C01835=1141.275,213.757,-64.467,-177.986,7.593,148.858
C01836=1141.271,214.006,-64.493,-177.983,7.596,148.857
C01837=1141.266,214.256,-64.518,-177.981,7.599,148.857
C01838=1141.261,214.504,-64.544,-177.977,7.602,148.857
C01839=1141.257,214.753,-64.569,-177.975,7.604,148.857
C01840=1141.253,215.001,-64.593,-177.972,7.607,148.857
C01841=1141.248,215.250,-64.619,-177.969,7.610,148.857
C01842=1141.243,215.498,-64.644,-177.966,7.612,148.856
C01843=1141.239,215.747,-64.670,-177.963,7.615,148.856
C01844=1141.234,215.995,-64.695,-177.961,7.617,148.856
C01845=1141.230,216.245,-64.720,-177.958,7.620,148.856
C01846=1141.225,216.494,-64.746,-177.955,7.623,148.856
C01847=1141.221,216.741,-64.770,-177.952,7.626,148.856
C01848=1141.217,216.991,-64.796,-177.950,7.628,148.856
C01849=1141.212,217.239,-64.821,-177.947,7.631,148.855
C01850=1141.208,217.488,-64.847,-177.944,7.633,148.855
C01851=1141.203,217.737,-64.872,-177.941,7.636,148.855
C01852=1141.198,217.985,-64.897,-177.938,7.639,148.855
C01853=1141.194,218.234,-64.923,-177.936,7.641,148.855
C01854=1141.189,218.482,-64.948,-177.933,7.644,148.854
C01855=1141.185,218.731,-64.974,-177.930,7.646,148.854
C01856=1141.181,218.980,-64.999,-177.927,7.649,148.854
C01857=1141.176,219.228,-65.024,-177.924,7.652,148.854
C01858=1141.172,219.477,-65.050,-177.922,7.654,148.854
C01859=1141.167,219.726,-65.076,-177.919,7.657,148.854
C01860=1141.162,219.974,-65.101,-177.916,7.660,148.854
C01861=1141.158,220.223,-65.127,-177.913,7.663,148.854
C01862=1141.154,220.472,-65.153,-177.911,7.666,148.853
C01863=1141.149,220.720,-65.177,-177.907,7.668,148.853
C01864=1141.145,220.969,-65.203,-177.905,7.670,148.853
C01865=1141.140,221.218,-65.229,-177.902,7.673,148.853
C01866=1141.136,221.466,-65.254,-177.899,7.676,148.853
C01867=1141.131,221.715,-65.280,-177.897,7.679,148.853
C01868=1141.127,221.964,-65.306,-177.894,7.682,148.853
C01869=1141.123,222.213,-65.332,-177.891,7.685,148.852
C01870=1141.118,222.461,-65.357,-177.888,7.687,148.852
C01871=1141.114,222.709,-65.383,-177.886,7.690,148.852
C01872=1141.109,222.959,-65.409,-177.883,7.692,148.852
C01873=1141.104,223.207,-65.434,-177.880,7.695,148.852
C01874=1141.100,223.456,-65.460,-177.877,7.698,148.852
C01875=1141.096,223.704,-65.486,-177.874,7.701,148.852
C01876=1141.091,223.953,-65.512,-177.872,7.703,148.851
C01877=1141.087,224.201,-65.537,-177.869,7.706,148.851
C01878=1141.083,224.449,-65.564,-177.866,7.709,148.851
C01879=1141.078,224.699,-65.590,-177.863,7.712,148.851
C01880=1141.074,224.947,-65.616,-177.860,7.714,148.851
C01881=1141.069,225.195,-65.641,-177.857,7.717,148.851
C01882=1141.064,225.444,-65.667,-177.854,7.720,148.851
C01883=1141.060,225.693,-65.693,-177.852,7.722,148.851
C01884=1141.055,225.942,-65.719,-177.849,7.725,148.850
C01885=1141.051,226.190,-65.745,-177.847,7.728,148.850
C01886=1141.047,226.438,-65.771,-177.843,7.731,148.850
C01887=1141.042,226.687,-65.796,-177.841,7.733,148.850
C01888=1141.037,226.936,-65.823,-177.838,7.736,148.850
C01889=1141.033,227.185,-65.849,-177.835,7.739,148.850
C01890=1141.029,227.433,-65.875,-177.833,7.741,148.850
C01891=1141.024,227.681,-65.900,-177.830,7.744,148.850
C01892=1141.019,227.931,-65.927,-177.827,7.747,148.850
C01893=1141.015,228.179,-65.953,-177.824,7.750,148.849
C01894=1141.011,228.428,-65.979,-177.821,7.753,148.849
C01895=1141.006,228.677,-66.005,-177.818,7.756,148.849
C01896=1141.002,228.925,-66.032,-177.815,7.759,148.849
C01897=1140.998,229.174,-66.058,-177.813,7.761,148.849
C01898=1140.993,229.422,-66.084,-177.810,7.764,148.849
C01899=1140.989,229.670,-66.110,-177.808,7.766,148.849
C01900=1140.984,229.919,-66.136,-177.805,7.769,148.849
C01901=1140.979,230.168,-66.162,-177.802,7.772,148.848
C01902=1140.976,230.416,-66.189,-177.799,7.775,148.848
C01903=1140.971,230.665,-66.214,-177.796,7.778,148.848
C01904=1140.967,230.914,-66.241,-177.793,7.781,148.848
C01905=1140.962,231.162,-66.267,-177.790,7.784,148.848
C01906=1140.958,231.411,-66.294,-177.788,7.786,148.848
C01907=1140.953,231.659,-66.320,-177.785,7.789,148.848
C01908=1140.949,231.907,-66.346,-177.783,7.791,148.848
C01909=1140.944,232.156,-66.372,-177.780,7.794,148.848
C01910=1140.940,232.405,-66.399,-177.777,7.797,148.847
C01911=1140.935,232.654,-66.425,-177.774,7.800,148.847
C01912=1140.931,232.902,-66.452,-177.771,7.803,148.847
C01913=1140.926,233.151,-66.478,-177.768,7.806,148.847
C01914=1140.922,233.399,-66.504,-177.765,7.809,148.847
C01915=1140.918,233.648,-66.532,-177.763,7.812,148.847
C01916=1140.914,233.896,-66.557,-177.760,7.814,148.847
C01917=1140.909,234.145,-66.584,-177.757,7.817,148.847
C01918=1140.905,234.394,-66.610,-177.754,7.820,148.847
C01919=1140.900,234.642,-66.637,-177.752,7.822,148.846
C01920=1140.896,234.890,-66.664,-177.749,7.825,148.846
C01921=1140.891,235.163,-66.692,-177.746,7.829,148.846
C01922=1140.886,235.434,-66.722,-177.743,7.832,148.846
C01923=1140.882,235.706,-66.751,-177.740,7.834,148.846
C01924=1140.877,235.978,-66.780,-177.736,7.838,148.846
C01925=1140.872,236.227,-66.806,-177.733,7.841,148.846
C01926=1140.868,236.475,-66.833,-177.731,7.843,148.846
C01927=1140.863,236.724,-66.860,-177.728,7.846,148.846
C01928=1140.859,236.972,-66.886,-177.726,7.849,148.846
C01929=1140.854,237.221,-66.913,-177.723,7.852,148.845
C01930=1140.850,237.469,-66.940,-177.720,7.855,148.845
C01931=1140.846,237.718,-66.966,-177.717,7.858,148.845
C01932=1140.841,237.966,-66.993,-177.714,7.861,148.845
C01933=1140.836,238.215,-67.020,-177.712,7.864,148.845
C01934=1140.832,238.463,-67.046,-177.709,7.867,148.845
C01935=1140.827,238.712,-67.073,-177.706,7.869,148.845
C01936=1140.823,238.961,-67.101,-177.703,7.872,148.845
C01937=1140.819,239.209,-67.127,-177.701,7.875,148.845
C01938=1140.815,239.458,-67.154,-177.698,7.878,148.845
C01939=1140.810,239.706,-67.181,-177.695,7.881,148.845
C01940=1140.806,239.954,-67.208,-177.692,7.884,148.845
C01941=1140.802,240.203,-67.235,-177.689,7.887,148.844
C01942=1140.797,240.451,-67.262,-177.687,7.890,148.844
C01943=1140.792,240.700,-67.289,-177.684,7.893,148.844
C01944=1140.788,240.948,-67.315,-177.681,7.896,148.844
C01945=1140.784,241.197,-67.342,-177.678,7.899,148.844
C01946=1140.780,241.446,-67.370,-177.675,7.902,148.844
C01947=1140.775,241.694,-67.397,-177.673,7.904,148.844
C01948=1140.771,241.943,-67.423,-177.670,7.907,148.844
C01949=1140.766,242.191,-67.450,-177.668,7.909,148.844
C01950=1140.762,242.440,-67.477,-177.665,7.912,148.844
C01951=1140.757,242.688,-67.505,-177.662,7.915,148.844
C01952=1140.752,242.937,-67.532,-177.659,7.918,148.844
C01953=1140.749,243.185,-67.558,-177.656,7.921,148.843
C01954=1140.744,243.434,-67.586,-177.654,7.924,148.843
C01955=1140.740,243.682,-67.613,-177.651,7.927,148.843
C01956=1140.735,243.930,-67.640,-177.648,7.930,148.843
C01957=1140.731,244.179,-67.667,-177.645,7.933,148.843
C01958=1140.727,244.428,-67.695,-177.642,7.936,148.843
C01959=1140.722,244.676,-67.722,-177.640,7.939,148.843
C01960=1140.718,244.925,-67.748,-177.637,7.942,148.843
C01961=1140.714,245.172,-67.776,-177.634,7.944,148.843
C01962=1140.709,245.421,-67.803,-177.631,7.947,148.843
C01963=1140.705,245.670,-67.831,-177.628,7.950,148.843
C01964=1140.700,245.919,-67.858,-177.626,7.953,148.843
C01965=1140.696,246.167,-67.885,-177.623,7.956,148.843
C01966=1140.691,246.415,-67.913,-177.620,7.959,148.843
C01967=1140.687,246.664,-67.940,-177.617,7.962,148.842
C01968=1140.683,246.913,-67.967,-177.614,7.965,148.842
C01969=1140.678,247.161,-67.995,-177.612,7.968,148.842
C01970=1140.674,247.409,-68.022,-177.609,7.971,148.842
C01971=1140.670,247.658,-68.050,-177.606,7.974,148.842
C01972=1140.665,247.906,-68.077,-177.603,7.977,148.842
C01973=1140.661,248.155,-68.104,-177.600,7.979,148.842
C01974=1140.656,248.403,-68.132,-177.598,7.982,148.842
C01975=1140.652,248.652,-68.159,-177.595,7.985,148.842
C01976=1140.648,248.900,-68.186,-177.592,7.989,148.842
C01977=1140.643,249.148,-68.214,-177.590,7.991,148.842
C01978=1140.639,249.397,-68.242,-177.587,7.994,148.842
C01979=1140.635,249.645,-68.269,-177.584,7.997,148.842
C01980=1140.630,249.894,-68.296,-177.581,8.000,148.842
C01981=1140.626,250.142,-68.324,-177.578,8.004,148.842
C01982=1140.622,250.391,-68.352,-177.575,8.007,148.842
C01983=1140.617,250.639,-68.379,-177.572,8.010,148.842
C01984=1140.613,250.887,-68.406,-177.570,8.013,148.841
C01985=1140.608,251.136,-68.435,-177.567,8.016,148.841
C01986=1140.604,251.385,-68.462,-177.564,8.019,148.841
C01987=1140.600,251.633,-68.490,-177.561,8.021,148.841
C01988=1140.596,251.881,-68.518,-177.559,8.025,148.841
C01989=1140.591,252.129,-68.545,-177.556,8.028,148.841
C01990=1140.587,252.378,-68.573,-177.553,8.031,148.841
C01991=1140.583,252.626,-68.601,-177.550,8.034,148.841
C01992=1140.577,252.875,-68.629,-177.548,8.036,148.841
C01993=1140.574,253.123,-68.657,-177.545,8.039,148.841
C01994=1140.569,253.372,-68.684,-177.542,8.042,148.841
C01995=1140.565,253.620,-68.712,-177.539,8.045,148.841
C01996=1140.561,253.868,-68.740,-177.536,8.048,148.841
C01997=1140.556,254.116,-68.768,-177.534,8.051,148.841
C01998=1140.552,254.366,-68.796,-177.531,8.054,148.841
C01999=1140.547,254.614,-68.824,-177.529,8.057,148.841
C02000=1140.544,254.862,-68.852,-177.526,8.060,148.841
C02001=1140.539,255.110,-68.879,-177.523,8.063,148.841
C02002=1140.534,255.359,-68.907,-177.520,8.066,148.841
C02003=1140.530,255.607,-68.935,-177.517,8.070,148.841
C02004=1140.526,255.855,-68.963,-177.514,8.073,148.841
C02005=1140.521,256.104,-68.992,-177.512,8.076,148.841
C02006=1140.517,256.352,-69.020,-177.509,8.079,148.841
C02007=1140.513,256.601,-69.047,-177.506,8.082,148.841
C02008=1140.508,256.849,-69.075,-177.503,8.085,148.840
C02009=1140.504,257.098,-69.103,-177.500,8.088,148.840
C02010=1140.500,257.346,-69.131,-177.498,8.090,148.840
C02011=1140.495,257.595,-69.160,-177.495,8.093,148.840
C02012=1140.491,257.843,-69.188,-177.493,8.097,148.840
C02013=1140.487,258.091,-69.216,-177.490,8.100,148.840
C02014=1140.482,258.339,-69.244,-177.487,8.102,148.840
C02015=1140.478,258.588,-69.272,-177.484,8.105,148.840
C02016=1140.474,258.836,-69.300,-177.481,8.109,148.840
C02017=1140.469,259.085,-69.329,-177.478,8.112,148.840
C02018=1140.465,259.333,-69.357,-177.476,8.115,148.840
C02019=1140.461,259.581,-69.385,-177.473,8.118,148.840
C02020=1140.456,259.829,-69.413,-177.470,8.121,148.840
C02021=1140.452,260.078,-69.441,-177.467,8.124,148.840
C02022=1140.447,260.326,-69.470,-177.464,8.127,148.840
C02023=1140.444,260.575,-69.498,-177.462,8.130,148.840
C02024=1140.439,260.823,-69.526,-177.459,8.133,148.840
C02025=1140.434,261.097,-69.557,-177.456,8.137,148.840
C02026=1140.429,261.371,-69.589,-177.453,8.140,148.840
C02027=1140.425,261.643,-69.620,-177.450,8.144,148.840
C02028=1140.420,261.918,-69.652,-177.447,8.146,148.840
C02029=1140.416,262.165,-69.679,-177.444,8.149,148.840
C02030=1140.411,262.414,-69.708,-177.441,8.153,148.840
C02031=1140.407,262.662,-69.736,-177.439,8.156,148.840
C02032=1140.403,262.911,-69.765,-177.436,8.159,148.840
C02033=1140.399,263.159,-69.794,-177.433,8.162,148.840
C02034=1140.394,263.407,-69.822,-177.430,8.165,148.840
C02035=1140.390,263.656,-69.850,-177.428,8.168,148.840
C02036=1140.385,263.903,-69.879,-177.425,8.171,148.840
C02037=1140.381,264.152,-69.907,-177.422,8.174,148.840
C02038=1140.377,264.401,-69.936,-177.419,8.178,148.840
C02039=1140.372,264.649,-69.964,-177.417,8.181,148.840
C02040=1140.368,264.897,-69.993,-177.414,8.184,148.840
C02041=1140.364,265.146,-70.022,-177.411,8.187,148.840
C02042=1140.359,265.394,-70.050,-177.408,8.190,148.840
C02043=1140.355,265.642,-70.079,-177.406,8.193,148.840
C02044=1140.351,265.891,-70.108,-177.403,8.196,148.840
C02045=1140.347,266.138,-70.136,-177.400,8.199,148.840
C02046=1140.342,266.387,-70.165,-177.397,8.203,148.840
C02047=1140.338,266.636,-70.194,-177.395,8.206,148.840
C02048=1140.334,266.883,-70.222,-177.392,8.209,148.840
C02049=1140.329,267.132,-70.251,-177.389,8.212,148.840
C02050=1140.325,267.380,-70.281,-177.386,8.215,148.840
C02051=1140.320,267.629,-70.309,-177.384,8.218,148.840
C02052=1140.317,267.877,-70.338,-177.381,8.221,148.840
C02053=1140.312,268.125,-70.367,-177.378,8.225,148.840
C02054=1140.308,268.374,-70.396,-177.375,8.228,148.840
C02055=1140.303,268.622,-70.424,-177.372,8.231,148.840
C02056=1140.299,268.870,-70.453,-177.370,8.234,148.840
C02057=1140.295,269.119,-70.482,-177.367,8.237,148.840
C02058=1140.291,269.367,-70.511,-177.365,8.240,148.840
C02059=1140.286,269.615,-70.540,-177.362,8.243,148.840
C02060=1140.282,269.863,-70.569,-177.358,8.247,148.840
C02061=1140.278,270.112,-70.597,-177.356,8.250,148.840
C02062=1140.274,270.360,-70.627,-177.353,8.253,148.840
C02063=1140.269,270.608,-70.656,-177.350,8.256,148.840
C02064=1140.264,270.857,-70.685,-177.348,8.259,148.840
C02065=1140.261,271.105,-70.714,-177.345,8.262,148.840
C02066=1140.257,271.353,-70.743,-177.342,8.266,148.840
C02067=1140.252,271.602,-70.772,-177.339,8.269,148.840
C02068=1140.247,271.849,-70.801,-177.337,8.272,148.840
C02069=1140.243,272.098,-70.830,-177.334,8.275,148.840
C02070=1140.239,272.346,-70.860,-177.331,8.278,148.840
C02071=1140.235,272.595,-70.888,-177.329,8.281,148.840
C02072=1140.231,272.843,-70.917,-177.326,8.285,148.840
C02073=1140.226,273.090,-70.946,-177.323,8.288,148.840
C02074=1140.222,273.339,-70.976,-177.320,8.291,148.840
C02075=1140.218,273.588,-71.005,-177.318,8.294,148.840
C02076=1140.213,273.836,-71.034,-177.315,8.297,148.840
C02077=1140.209,274.084,-71.063,-177.312,8.301,148.840
C02078=1140.205,274.332,-71.093,-177.309,8.304,148.840
C02079=1140.201,274.581,-71.122,-177.306,8.307,148.840
C02080=1140.196,274.828,-71.151,-177.304,8.310,148.840
C02081=1140.192,275.076,-71.181,-177.301,8.313,148.840
C02082=1140.187,275.325,-71.210,-177.298,8.316,148.840
C02083=1140.183,275.574,-71.239,-177.296,8.320,148.840
C02084=1140.179,275.822,-71.269,-177.293,8.323,148.840
C02085=1140.175,276.070,-71.298,-177.290,8.326,148.840
C02086=1140.171,276.318,-71.327,-177.288,8.329,148.840
C02087=1140.167,276.567,-71.357,-177.285,8.332,148.840
C02088=1140.162,276.815,-71.386,-177.281,8.336,148.840
C02089=1140.158,277.063,-71.416,-177.279,8.339,148.841
C02090=1140.153,277.311,-71.445,-177.276,8.342,148.840
C02091=1140.149,277.559,-71.474,-177.274,8.345,148.841
C02092=1140.145,277.807,-71.504,-177.271,8.349,148.841
C02093=1140.141,278.056,-71.533,-177.268,8.352,148.841
C02094=1140.137,278.304,-71.563,-177.265,8.355,148.841
C02095=1140.133,278.552,-71.592,-177.263,8.358,148.841
C02096=1140.129,278.800,-71.622,-177.260,8.361,148.841
C02097=1140.124,279.048,-71.652,-177.257,8.365,148.841
C02098=1140.120,279.297,-71.682,-177.254,8.368,148.841
C02099=1140.115,279.545,-71.711,-177.252,8.371,148.841
C02100=1140.111,279.793,-71.741,-177.249,8.374,148.841
C02101=1140.107,280.041,-71.770,-177.247,8.377,148.841
C02102=1140.103,280.290,-71.800,-177.243,8.381,148.841
C02103=1140.099,280.537,-71.830,-177.241,8.384,148.841
C02104=1140.094,280.786,-71.860,-177.238,8.387,148.841
C02105=1140.090,281.034,-71.889,-177.235,8.390,148.841
C02106=1140.086,281.282,-71.919,-177.233,8.394,148.841
C02107=1140.082,281.530,-71.949,-177.230,8.397,148.841
C02108=1140.078,281.778,-71.978,-177.227,8.401,148.841
C02109=1140.073,282.027,-72.008,-177.225,8.403,148.841
C02110=1140.068,282.275,-72.038,-177.222,8.408,148.842
C02111=1140.065,282.523,-72.068,-177.219,8.410,148.841
C02112=1140.060,282.771,-72.098,-177.216,8.413,148.841
C02113=1140.056,283.020,-72.128,-177.214,8.417,148.842
C02114=1140.052,283.267,-72.158,-177.210,8.420,148.842
C02115=1140.047,283.516,-72.187,-177.208,8.424,148.842
C02116=1140.043,283.764,-72.217,-177.205,8.427,148.842
C02117=1140.039,284.012,-72.247,-177.203,8.430,148.842
C02118=1140.035,284.261,-72.277,-177.200,8.434,148.842
C02119=1140.031,284.508,-72.307,-177.197,8.437,148.842
C02120=1140.026,284.757,-72.337,-177.194,8.440,148.842
C02121=1140.022,285.005,-72.368,-177.192,8.443,148.842
C02122=1140.018,285.253,-72.397,-177.189,8.447,148.842
C02123=1140.014,285.501,-72.428,-177.186,8.450,148.842
C02124=1140.009,285.749,-72.457,-177.184,8.453,148.842
C02125=1140.005,285.997,-72.488,-177.181,8.456,148.842
C02126=1140.001,286.245,-72.518,-177.178,8.460,148.842
C02127=1139.997,286.493,-72.548,-177.176,8.463,148.843
C02128=1139.992,286.742,-72.578,-177.173,8.466,148.843
C02129=1139.988,287.017,-72.611,-177.170,8.470,148.843
C02130=1139.983,287.293,-72.644,-177.166,8.474,148.843
C02131=1139.978,287.568,-72.678,-177.164,8.477,148.843
C02132=1139.974,287.844,-72.712,-177.161,8.481,148.843
C02133=1139.969,288.092,-72.742,-177.158,8.484,148.843
C02134=1139.965,288.340,-72.772,-177.155,8.488,148.843
C02135=1139.961,288.589,-72.803,-177.153,8.491,148.843
C02136=1139.957,288.837,-72.833,-177.150,8.494,148.843
C02137=1139.952,289.085,-72.864,-177.147,8.498,148.843
C02138=1139.949,289.332,-72.894,-177.144,8.501,148.843
C02139=1139.944,289.581,-72.924,-177.142,8.504,148.844
C02140=1139.940,289.829,-72.954,-177.139,8.507,148.843
C02141=1139.936,290.077,-72.985,-177.136,8.511,148.844
C02142=1139.932,290.325,-73.015,-177.133,8.514,148.844
C02143=1139.927,290.574,-73.045,-177.131,8.518,148.844
C02144=1139.923,290.821,-73.075,-177.128,8.522,148.844
C02145=1139.919,291.070,-73.107,-177.125,8.525,148.844
C02146=1139.915,291.318,-73.137,-177.123,8.528,148.844
C02147=1139.911,291.565,-73.168,-177.120,8.532,148.844
C02148=1139.906,291.814,-73.197,-177.117,8.535,148.844
C02149=1139.902,292.062,-73.228,-177.114,8.538,148.844
C02150=1139.898,292.310,-73.259,-177.112,8.541,148.844
C02151=1139.894,292.558,-73.289,-177.109,8.545,148.845
C02152=1139.889,292.806,-73.320,-177.106,8.548,148.845
C02153=1139.886,293.054,-73.350,-177.104,8.551,148.845
C02154=1139.881,293.302,-73.381,-177.101,8.555,148.845
C02155=1139.877,293.550,-73.412,-177.098,8.558,148.845
C02156=1139.874,293.799,-73.442,-177.096,8.562,148.845
C02157=1139.869,294.047,-73.473,-177.093,8.565,148.845
C02158=1139.864,294.294,-73.504,-177.090,8.569,148.845
C02159=1139.861,294.543,-73.534,-177.088,8.571,148.845
C02160=1139.856,294.791,-73.565,-177.085,8.576,148.845
C02161=1139.852,295.039,-73.596,-177.082,8.579,148.846
C02162=1139.848,295.286,-73.626,-177.080,8.582,148.846
C02163=1139.844,295.535,-73.657,-177.077,8.586,148.846
C02164=1139.839,295.783,-73.688,-177.074,8.589,148.846
C02165=1139.835,296.032,-73.719,-177.071,8.592,148.846
C02166=1139.831,296.279,-73.749,-177.069,8.596,148.846
C02167=1139.827,296.527,-73.780,-177.066,8.599,148.846
C02168=1139.823,296.776,-73.811,-177.063,8.602,148.846
C02169=1139.818,297.023,-73.843,-177.060,8.606,148.846
C02170=1139.815,297.271,-73.873,-177.058,8.609,148.846
C02171=1139.811,297.520,-73.904,-177.055,8.612,148.847
C02172=1139.806,297.768,-73.935,-177.052,8.617,148.847
C02173=1139.801,298.016,-73.966,-177.050,8.620,148.847
C02174=1139.797,298.264,-73.997,-177.047,8.623,148.847
C02175=1139.794,298.511,-74.028,-177.044,8.627,148.847
C02176=1139.790,298.760,-74.059,-177.042,8.630,148.847
C02177=1139.785,299.008,-74.089,-177.039,8.633,148.847
C02178=1139.781,299.256,-74.120,-177.036,8.637,148.847
C02179=1139.777,299.504,-74.152,-177.034,8.640,148.848
C02180=1139.772,299.752,-74.183,-177.031,8.643,148.848
C02181=1139.768,300.000,-74.214,-177.028,8.647,148.848
C02182=1139.764,300.248,-74.245,-177.026,8.651,148.848
C02183=1139.761,300.496,-74.276,-177.023,8.654,148.848
C02184=1139.756,300.744,-74.307,-177.020,8.658,148.848
C02185=1139.752,300.992,-74.339,-177.018,8.661,148.848
C02186=1139.748,301.240,-74.369,-177.015,8.665,148.848
C02187=1139.743,301.487,-74.401,-177.012,8.668,148.849
C02188=1139.739,301.736,-74.432,-177.010,8.671,148.849
C02189=1139.735,301.984,-74.463,-177.007,8.675,148.849
C02190=1139.731,302.232,-74.495,-177.004,8.678,148.849
C02191=1139.726,302.480,-74.525,-177.001,8.682,148.849
C02192=1139.723,302.728,-74.557,-176.999,8.685,148.849
C02193=1139.718,302.976,-74.588,-176.997,8.689,148.849
C02194=1139.714,303.224,-74.620,-176.993,8.692,148.849
C02195=1139.710,303.472,-74.651,-176.991,8.696,148.850
C02196=1139.706,303.720,-74.682,-176.988,8.699,148.850
C02197=1139.701,303.968,-74.713,-176.986,8.703,148.850
C02198=1139.698,304.216,-74.745,-176.983,8.706,148.850
C02199=1139.693,304.464,-74.776,-176.980,8.710,148.850
C02200=1139.689,304.712,-74.808,-176.977,8.713,148.850
C02201=1139.685,304.959,-74.839,-176.975,8.717,148.851
C02202=1139.680,305.208,-74.871,-176.972,8.720,148.851
C02203=1139.676,305.456,-74.902,-176.969,8.724,148.851
C02204=1139.672,305.704,-74.934,-176.967,8.728,148.851
C02205=1139.668,305.952,-74.965,-176.964,8.731,148.851
C02206=1139.664,306.200,-74.997,-176.962,8.734,148.851
C02207=1139.660,306.448,-75.029,-176.958,8.738,148.851
C02208=1139.656,306.696,-75.059,-176.956,8.741,148.852
C02209=1139.652,306.944,-75.091,-176.953,8.745,148.852
C02210=1139.647,307.191,-75.123,-176.951,8.749,148.852
C02211=1139.643,307.440,-75.154,-176.949,8.752,148.852
C02212=1139.639,307.688,-75.186,-176.945,8.756,148.852
C02213=1139.635,307.935,-75.218,-176.943,8.759,148.852
C02214=1139.631,308.183,-75.250,-176.940,8.763,148.852
C02215=1139.628,308.432,-75.281,-176.938,8.766,148.853
C02216=1139.622,308.680,-75.313,-176.935,8.770,148.853
C02217=1139.618,308.928,-75.345,-176.932,8.773,148.853
C02218=1139.614,309.175,-75.376,-176.929,8.776,148.853
C02219=1139.610,309.423,-75.408,-176.927,8.780,148.853
C02220=1139.606,309.672,-75.440,-176.924,8.784,148.853
C02221=1139.602,309.919,-75.472,-176.921,8.788,148.854
C02222=1139.598,310.167,-75.504,-176.919,8.791,148.854
C02223=1139.594,310.415,-75.536,-176.916,8.795,148.854
C02224=1139.589,310.663,-75.568,-176.914,8.798,148.854
C02225=1139.586,310.911,-75.600,-176.911,8.802,148.854
C02226=1139.582,311.159,-75.631,-176.908,8.805,148.854
C02227=1139.577,311.407,-75.662,-176.906,8.809,148.855
C02228=1139.573,311.655,-75.695,-176.903,8.813,148.855
C02229=1139.569,311.903,-75.726,-176.900,8.816,148.855
C02230=1139.565,312.150,-75.759,-176.897,8.820,148.855
C02231=1139.561,312.398,-75.791,-176.895,8.823,148.855
C02232=1139.557,312.646,-75.823,-176.892,8.827,148.856
C02233=1139.552,312.925,-75.858,-176.890,8.831,148.856
C02234=1139.547,313.202,-75.894,-176.887,8.835,148.856
C02235=1139.543,313.481,-75.931,-176.884,8.838,148.856
C02236=1139.538,313.758,-75.966,-176.881,8.843,148.856
C02237=1139.534,314.007,-75.999,-176.878,8.847,148.857
C02238=1139.530,314.254,-76.030,-176.875,8.850,148.857
C02239=1139.526,314.501,-76.063,-176.872,8.854,148.857
C02240=1139.522,314.750,-76.095,-176.870,8.857,148.857
C02241=1139.518,314.998,-76.127,-176.867,8.861,148.857
C02242=1139.513,315.245,-76.159,-176.865,8.864,148.858
C02243=1139.509,315.493,-76.191,-176.862,8.869,148.858
C02244=1139.505,315.741,-76.224,-176.860,8.872,148.858
C02245=1139.502,315.989,-76.256,-176.857,8.876,148.858
C02246=1139.497,316.238,-76.288,-176.854,8.879,148.858
C02247=1139.493,316.485,-76.320,-176.851,8.883,148.859
C02248=1139.489,316.733,-76.353,-176.849,8.886,148.859
C02249=1139.485,316.981,-76.385,-176.846,8.891,148.859
C02250=1139.481,317.229,-76.417,-176.844,8.894,148.859
C02251=1139.477,317.476,-76.450,-176.841,8.898,148.859
C02252=1139.472,317.724,-76.482,-176.838,8.901,148.860
C02253=1139.469,317.971,-76.514,-176.836,8.904,148.860
C02254=1139.464,318.220,-76.547,-176.833,8.908,148.860
C02255=1139.461,318.468,-76.579,-176.831,8.912,148.860
C02256=1139.456,318.716,-76.612,-176.828,8.916,148.860
C02257=1139.453,318.964,-76.644,-176.826,8.919,148.861
C02258=1139.449,319.211,-76.677,-176.823,8.923,148.861
C02259=1139.444,319.459,-76.709,-176.820,8.926,148.861
C02260=1139.440,319.706,-76.741,-176.817,8.930,148.861
C02261=1139.436,319.955,-76.774,-176.815,8.934,148.861
C02262=1139.432,320.202,-76.806,-176.812,8.938,148.862
C02263=1139.428,320.451,-76.839,-176.810,8.941,148.862
C02264=1139.424,320.698,-76.872,-176.807,8.945,148.862
C02265=1139.420,320.946,-76.904,-176.804,8.948,148.862
C02266=1139.416,321.194,-76.937,-176.802,8.952,148.862
C02267=1139.411,321.442,-76.970,-176.799,8.956,148.863
C02268=1139.408,321.690,-77.002,-176.796,8.960,148.863
C02269=1139.404,321.938,-77.035,-176.793,8.964,148.863
C02270=1139.399,322.186,-77.068,-176.791,8.967,148.863
C02271=1139.395,322.433,-77.100,-176.788,8.971,148.863
C02272=1139.391,322.681,-77.132,-176.786,8.974,148.864
C02273=1139.387,322.929,-77.165,-176.783,8.979,148.864
C02274=1139.383,323.176,-77.198,-176.780,8.982,148.864
C02275=1139.379,323.424,-77.230,-176.778,8.986,148.864
C02276=1139.375,323.672,-77.264,-176.776,8.989,148.865
C02277=1139.371,323.920,-77.297,-176.773,8.993,148.865
C02278=1139.367,324.167,-77.329,-176.770,8.997,148.865
C02279=1139.363,324.416,-77.362,-176.767,9.001,148.865
C02280=1139.359,324.663,-77.395,-176.765,9.004,148.866
C02281=1139.355,324.911,-77.428,-176.762,9.008,148.866
C02282=1139.350,325.159,-77.461,-176.760,9.011,148.866
C02283=1139.347,325.406,-77.494,-176.757,9.015,148.866
C02284=1139.343,325.655,-77.526,-176.755,9.019,148.866
C02285=1139.338,325.902,-77.559,-176.752,9.023,148.867
C02286=1139.334,326.150,-77.593,-176.749,9.027,148.867
C02287=1139.330,326.398,-77.626,-176.747,9.030,148.867
C02288=1139.326,326.646,-77.659,-176.744,9.035,148.867
C02289=1139.322,326.893,-77.692,-176.742,9.038,148.868
C02290=1139.319,327.141,-77.725,-176.739,9.042,148.868
C02291=1139.314,327.388,-77.758,-176.736,9.045,148.868
C02292=1139.311,327.637,-77.791,-176.734,9.050,148.869
C02293=1139.307,327.885,-77.824,-176.731,9.053,148.869
C02294=1139.302,328.133,-77.857,-176.728,9.057,148.869
C02295=1139.298,328.381,-77.890,-176.726,9.061,148.869
C02296=1139.294,328.628,-77.923,-176.723,9.064,148.869
C02297=1139.290,328.876,-77.957,-176.720,9.068,148.870
C02298=1139.286,329.123,-77.990,-176.718,9.072,148.870
C02299=1139.282,329.371,-78.023,-176.715,9.076,148.870
C02300=1139.278,329.619,-78.057,-176.713,9.079,148.870
C02301=1139.274,329.866,-78.090,-176.710,9.083,148.871
C02302=1139.269,330.114,-78.123,-176.708,9.086,148.871
C02303=1139.265,330.362,-78.156,-176.705,9.091,148.871
C02304=1139.262,330.610,-78.189,-176.702,9.095,148.872
C02305=1139.258,330.858,-78.223,-176.700,9.098,148.872
C02306=1139.254,331.106,-78.256,-176.697,9.102,148.872
C02307=1139.250,331.353,-78.290,-176.695,9.106,148.872
C02308=1139.246,331.601,-78.323,-176.692,9.110,148.873
C02309=1139.241,331.848,-78.356,-176.689,9.114,148.873
C02310=1139.237,332.096,-78.389,-176.687,9.117,148.873
C02311=1139.234,332.345,-78.423,-176.684,9.121,148.873
C02312=1139.230,332.592,-78.457,-176.682,9.125,148.874
C02313=1139.226,332.839,-78.490,-176.679,9.129,148.874
C02314=1139.222,333.087,-78.523,-176.677,9.132,148.874
C02315=1139.217,333.335,-78.557,-176.674,9.136,148.874
C02316=1139.214,333.583,-78.591,-176.671,9.141,148.875
C02317=1139.209,333.831,-78.624,-176.669,9.144,148.875
C02318=1139.205,334.078,-78.657,-176.666,9.148,148.875
C02319=1139.201,334.325,-78.691,-176.664,9.152,148.876
C02320=1139.197,334.573,-78.724,-176.661,9.156,148.876
C02321=1139.194,334.822,-78.758,-176.658,9.160,148.876
C02322=1139.189,335.069,-78.792,-176.656,9.163,148.876
C02323=1139.185,335.317,-78.825,-176.654,9.167,148.877
C02324=1139.181,335.564,-78.859,-176.651,9.171,148.877
C02325=1139.178,335.812,-78.893,-176.648,9.175,148.877
C02326=1139.174,336.059,-78.927,-176.646,9.179,148.878
C02327=1139.169,336.307,-78.960,-176.643,9.182,148.878
C02328=1139.165,336.555,-78.994,-176.641,9.186,148.878
C02329=1139.162,336.803,-79.028,-176.638,9.191,148.878
C02330=1139.158,337.050,-79.062,-176.636,9.194,148.879
C02331=1139.153,337.298,-79.095,-176.633,9.198,148.879
C02332=1139.149,337.545,-79.129,-176.630,9.203,148.879
C02333=1139.146,337.794,-79.163,-176.628,9.206,148.880
C02334=1139.142,338.041,-79.197,-176.625,9.210,148.880
C02335=1139.137,338.289,-79.230,-176.623,9.213,148.880
C02336=1139.134,338.537,-79.265,-176.620,9.217,148.880
C02337=1139.129,338.817,-79.303,-176.617,9.222,148.881
C02338=1139.124,339.098,-79.342,-176.614,9.227,148.881
C02339=1139.119,339.379,-79.380,-176.611,9.231,148.881
C02340=1139.115,339.659,-79.419,-176.609,9.235,148.882
C02341=1139.111,339.907,-79.453,-176.606,9.239,148.882
C02342=1139.107,340.155,-79.486,-176.603,9.243,148.882
C02343=1139.103,340.402,-79.520,-176.601,9.247,148.883
C02344=1139.099,340.650,-79.555,-176.598,9.251,148.883
C02345=1139.095,340.898,-79.588,-176.596,9.255,148.883
C02346=1139.091,341.145,-79.622,-176.593,9.259,148.884
C02347=1139.088,341.393,-79.657,-176.590,9.263,148.884
C02348=1139.083,341.640,-79.691,-176.588,9.266,148.884
C02349=1139.079,341.888,-79.724,-176.585,9.270,148.885
C02350=1139.075,342.136,-79.759,-176.583,9.275,148.885
C02351=1139.071,342.383,-79.793,-176.580,9.278,148.885
C02352=1139.066,342.631,-79.827,-176.578,9.282,148.886
C02353=1139.063,342.878,-79.862,-176.575,9.286,148.886
C02354=1139.059,343.126,-79.896,-176.573,9.290,148.886
C02355=1139.055,343.374,-79.930,-176.570,9.294,148.886
C02356=1139.051,343.621,-79.965,-176.567,9.298,148.887
C02357=1139.047,343.869,-79.998,-176.565,9.302,148.887
C02358=1139.043,344.117,-80.033,-176.562,9.306,148.887
C02359=1139.039,344.364,-80.067,-176.560,9.310,148.888
C02360=1139.035,344.612,-80.101,-176.558,9.313,148.888
C02361=1139.031,344.859,-80.135,-176.555,9.318,148.888
C02362=1139.027,345.107,-80.170,-176.552,9.322,148.889
C02363=1139.023,345.355,-80.204,-176.550,9.326,148.889
C02364=1139.019,345.602,-80.238,-176.547,9.330,148.889
C02365=1139.015,345.850,-80.273,-176.544,9.334,148.890
C02366=1139.011,346.097,-80.307,-176.542,9.337,148.890
C02367=1139.007,346.345,-80.342,-176.539,9.341,148.890
C02368=1139.003,346.592,-80.377,-176.537,9.346,148.891
C02369=1138.999,346.840,-80.411,-176.535,9.349,148.891
C02370=1138.995,347.087,-80.446,-176.532,9.353,148.891
C02371=1138.992,347.335,-80.480,-176.530,9.358,148.892
C02372=1138.987,347.583,-80.515,-176.527,9.362,148.892
C02373=1138.983,347.831,-80.549,-176.525,9.365,148.892
C02374=1138.979,348.078,-80.583,-176.522,9.369,148.893
C02375=1138.976,348.325,-80.619,-176.519,9.374,148.893
C02376=1138.971,348.573,-80.653,-176.517,9.377,148.893
C02377=1138.968,348.821,-80.688,-176.514,9.381,148.894
C02378=1138.963,349.068,-80.722,-176.512,9.386,148.894
C02379=1138.960,349.315,-80.758,-176.510,9.389,148.894
C02380=1138.956,349.564,-80.792,-176.507,9.393,148.895
C02381=1138.952,349.811,-80.826,-176.504,9.398,148.895
C02382=1138.948,350.059,-80.861,-176.501,9.402,148.895
C02383=1138.944,350.306,-80.896,-176.499,9.405,148.896
C02384=1138.940,350.554,-80.931,-176.497,9.410,148.896
C02385=1138.936,350.801,-80.965,-176.494,9.414,148.897
C02386=1138.932,351.048,-81.001,-176.491,9.418,148.897
C02387=1138.928,351.296,-81.035,-176.489,9.421,148.897
C02388=1138.924,351.544,-81.070,-176.486,9.426,148.898
C02389=1138.921,351.791,-81.105,-176.484,9.430,148.898
C02390=1138.916,352.038,-81.139,-176.482,9.433,148.898
C02391=1138.912,352.286,-81.175,-176.479,9.438,148.899
C02392=1138.908,352.534,-81.210,-176.476,9.442,148.899
C02393=1138.904,352.781,-81.245,-176.474,9.446,148.899
C02394=1138.900,353.029,-81.280,-176.471,9.449,148.900
C02395=1138.897,353.276,-81.315,-176.469,9.454,148.900
C02396=1138.893,353.524,-81.349,-176.466,9.458,148.901
C02397=1138.889,353.771,-81.385,-176.463,9.462,148.901
C02398=1138.884,354.019,-81.419,-176.461,9.466,148.901
C02399=1138.881,354.266,-81.455,-176.459,9.470,148.902
C02400=1138.877,354.514,-81.489,-176.456,9.474,148.902
C02401=1138.873,354.762,-81.525,-176.454,9.479,148.902
C02402=1138.869,355.008,-81.560,-176.452,9.482,148.903
C02403=1138.865,355.257,-81.595,-176.449,9.486,148.903
C02404=1138.861,355.504,-81.631,-176.446,9.491,148.903
C02405=1138.857,355.751,-81.664,-176.443,9.495,148.904
C02406=1138.854,355.999,-81.700,-176.441,9.498,148.904
C02407=1138.850,356.246,-81.736,-176.439,9.503,148.905
C02408=1138.846,356.493,-81.771,-176.436,9.507,148.905
C02409=1138.842,356.741,-81.806,-176.433,9.511,148.905
C02410=1138.838,356.989,-81.841,-176.431,9.515,148.906
C02411=1138.835,357.236,-81.877,-176.429,9.519,148.906
C02412=1138.830,357.484,-81.911,-176.426,9.523,148.906
C02413=1138.826,357.731,-81.947,-176.423,9.528,148.907
C02414=1138.823,357.979,-81.982,-176.421,9.532,148.907
C02415=1138.819,358.226,-82.018,-176.419,9.535,148.908
C02416=1138.815,358.473,-82.053,-176.416,9.540,148.908
C02417=1138.810,358.721,-82.089,-176.414,9.544,148.908
C02418=1138.806,358.969,-82.124,-176.411,9.548,148.909
C02419=1138.803,359.216,-82.159,-176.408,9.552,148.909
C02420=1138.798,359.463,-82.195,-176.406,9.556,148.910
C02421=1138.795,359.711,-82.230,-176.403,9.560,148.910
C02422=1138.791,359.958,-82.266,-176.401,9.564,148.910
C02423=1138.787,360.206,-82.301,-176.398,9.569,148.911
C02424=1138.784,360.453,-82.337,-176.396,9.573,148.911
C02425=1138.780,360.700,-82.372,-176.393,9.577,148.911
C02426=1138.776,360.947,-82.408,-176.390,9.582,148.912
C02427=1138.771,361.195,-82.444,-176.388,9.585,148.912
C02428=1138.768,361.443,-82.479,-176.385,9.589,148.913
C02429=1138.764,361.690,-82.515,-176.383,9.594,148.913
C02430=1138.760,361.938,-82.550,-176.380,9.598,148.914
C02431=1138.757,362.185,-82.586,-176.377,9.602,148.914
C02432=1138.753,362.432,-82.621,-176.375,9.606,148.914
C02433=1138.748,362.680,-82.657,-176.372,9.611,148.915
C02434=1138.744,362.927,-82.693,-176.370,9.615,148.915
C02435=1138.741,363.175,-82.728,-176.367,9.619,148.915
C02436=1138.737,363.422,-82.764,-176.364,9.624,148.916
C02437=1138.734,363.669,-82.800,-176.362,9.628,148.916
C02438=1138.729,363.917,-82.836,-176.359,9.632,148.917
C02439=1138.726,364.164,-82.872,-176.357,9.636,148.917
C02440=1138.722,364.412,-82.907,-176.355,9.640,148.917
C02441=1138.717,364.696,-82.949,-176.351,9.645,148.918
C02442=1138.713,364.980,-82.990,-176.348,9.650,148.918
C02443=1138.709,365.263,-83.031,-176.345,9.655,148.919
C02444=1138.704,365.548,-83.072,-176.342,9.660,148.919
C02445=1138.700,365.794,-83.108,-176.340,9.664,148.920
C02446=1138.696,366.042,-83.143,-176.337,9.669,148.920
C02447=1138.692,366.289,-83.180,-176.334,9.673,148.920
C02448=1138.688,366.537,-83.216,-176.332,9.677,148.921
C02449=1138.685,366.784,-83.251,-176.329,9.681,148.921
C02450=1138.681,367.031,-83.288,-176.326,9.685,148.922
C02451=1138.677,367.279,-83.323,-176.324,9.690,148.922
C02452=1138.673,367.526,-83.360,-176.321,9.694,148.923
C02453=1138.669,367.773,-83.396,-176.319,9.699,148.923
C02454=1138.666,368.021,-83.431,-176.316,9.703,148.923
C02455=1138.662,368.268,-83.468,-176.313,9.707,148.924
C02456=1138.658,368.516,-83.504,-176.311,9.711,148.924
C02457=1138.654,368.763,-83.541,-176.308,9.716,148.925
C02458=1138.650,369.010,-83.576,-176.305,9.720,148.925
C02459=1138.646,369.257,-83.613,-176.303,9.724,148.925
C02460=1138.642,369.505,-83.649,-176.300,9.729,148.926
C02461=1138.638,369.752,-83.686,-176.297,9.733,148.926
C02462=1138.635,370.000,-83.721,-176.295,9.737,148.927
C02463=1138.630,370.247,-83.758,-176.292,9.741,148.927
C02464=1138.627,370.494,-83.794,-176.290,9.746,148.928
C02465=1138.623,370.742,-83.830,-176.287,9.750,148.928
C02466=1138.619,370.988,-83.867,-176.284,9.754,148.928
C02467=1138.615,371.236,-83.903,-176.282,9.759,148.929
C02468=1138.612,371.483,-83.939,-176.279,9.763,148.929
C02469=1138.608,371.731,-83.976,-176.277,9.767,148.930
C02470=1138.604,371.979,-84.012,-176.274,9.771,148.930
C02471=1138.600,372.226,-84.049,-176.271,9.776,148.930
C02472=1138.596,372.473,-84.086,-176.269,9.780,148.931
C02473=1138.593,372.720,-84.122,-176.267,9.784,148.931
C02474=1138.589,372.968,-84.158,-176.264,9.788,148.932
C02475=1138.585,373.214,-84.194,-176.261,9.792,148.932
C02476=1138.581,373.462,-84.231,-176.259,9.797,148.932
C02477=1138.577,373.709,-84.268,-176.256,9.801,148.933
C02478=1138.573,373.956,-84.303,-176.254,9.805,148.933
C02479=1138.570,374.204,-84.341,-176.252,9.809,148.934
C02480=1138.566,374.451,-84.378,-176.249,9.813,148.934
C02481=1138.562,374.698,-84.414,-176.247,9.818,148.935
C02482=1138.558,374.945,-84.451,-176.244,9.821,148.935
C02483=1138.554,375.193,-84.487,-176.242,9.825,148.935
C02484=1138.551,375.440,-84.524,-176.239,9.830,148.936
C02485=1138.546,375.687,-84.560,-176.237,9.833,148.936
C02486=1138.543,375.935,-84.597,-176.235,9.838,148.937
C02487=1138.540,376.182,-84.633,-176.232,9.842,148.937
C02488=1138.535,376.429,-84.670,-176.230,9.846,148.938
C02489=1138.531,376.677,-84.707,-176.228,9.850,148.938
C02490=1138.527,376.924,-84.744,-176.226,9.853,148.939
C02491=1138.525,377.171,-84.781,-176.223,9.858,148.939
C02492=1138.520,377.418,-84.817,-176.222,9.861,148.939
C02493=1138.516,377.666,-84.854,-176.220,9.865,148.940
C02494=1138.512,377.913,-84.891,-176.218,9.870,148.940
C02495=1138.508,378.160,-84.928,-176.216,9.873,148.941
C02496=1138.505,378.408,-84.965,-176.214,9.877,148.941
C02497=1138.501,378.655,-85.002,-176.211,9.881,148.942
C02498=1138.498,378.901,-85.039,-176.209,9.885,148.942
C02499=1138.493,379.149,-85.076,-176.207,9.888,148.943
C02500=1138.489,379.396,-85.113,-176.206,9.892,148.943
C02501=1138.486,379.644,-85.150,-176.204,9.896,148.944
C02502=1138.482,379.891,-85.186,-176.202,9.899,148.944
C02503=1138.478,380.138,-85.223,-176.200,9.903,148.945
C02504=1138.474,380.385,-85.260,-176.198,9.907,148.945
C02505=1138.471,380.632,-85.298,-176.197,9.911,148.946
C02506=1138.467,380.879,-85.335,-176.195,9.914,148.946
C02507=1138.463,381.127,-85.372,-176.194,9.917,148.947
C02508=1138.459,381.374,-85.409,-176.192,9.921,148.947
C02509=1138.456,381.621,-85.445,-176.191,9.925,148.948
C02510=1138.452,381.868,-85.483,-176.189,9.927,148.948
C02511=1138.448,382.115,-85.520,-176.188,9.931,148.949
C02512=1138.445,382.363,-85.557,-176.187,9.934,148.949
C02513=1138.441,382.610,-85.594,-176.185,9.938,148.950
C02514=1138.437,382.857,-85.631,-176.184,9.941,148.950
C02515=1138.433,383.105,-85.668,-176.183,9.944,148.951
C02516=1138.429,383.352,-85.705,-176.181,9.948,148.951
C02517=1138.425,383.598,-85.743,-176.181,9.951,148.952
C02518=1138.421,383.846,-85.780,-176.180,9.954,148.952
C02519=1138.418,384.094,-85.817,-176.179,9.957,148.953
C02520=1138.414,384.341,-85.854,-176.178,9.960,148.954
C02521=1138.410,384.587,-85.891,-176.177,9.963,148.954
C02522=1138.406,384.835,-85.929,-176.176,9.966,148.955
C02523=1138.403,385.082,-85.966,-176.176,9.969,148.955
C02524=1138.399,385.329,-86.003,-176.175,9.972,148.956
C02525=1138.395,385.577,-86.040,-176.174,9.975,148.956
C02526=1138.391,385.823,-86.078,-176.174,9.978,148.957
C02527=1138.387,386.071,-86.115,-176.173,9.981,148.958
C02528=1138.384,386.318,-86.151,-176.173,9.983,148.958
C02529=1138.381,386.565,-86.189,-176.173,9.986,148.959
C02530=1138.377,386.812,-86.226,-176.173,9.989,148.960
C02531=1138.373,387.059,-86.264,-176.173,9.991,148.960
C02532=1138.369,387.306,-86.301,-176.173,9.994,148.961
C02533=1138.365,387.554,-86.337,-176.172,9.996,148.962
C02534=1138.362,387.801,-86.375,-176.172,9.999,148.962
C02535=1138.358,388.048,-86.412,-176.172,10.001,148.963
C02536=1138.354,388.295,-86.450,-176.173,10.004,148.964
C02537=1138.350,388.543,-86.488,-176.173,10.006,148.964
C02538=1138.346,388.789,-86.525,-176.173,10.009,148.965
C02539=1138.343,389.037,-86.562,-176.173,10.012,148.966
C02540=1138.339,389.284,-86.599,-176.173,10.014,148.966
C02541=1138.335,389.531,-86.637,-176.173,10.017,148.967
C02542=1138.331,389.779,-86.674,-176.174,10.018,148.968
C02543=1138.327,390.025,-86.712,-176.174,10.021,148.969
C02544=1138.323,390.273,-86.749,-176.174,10.024,148.969
C02545=1138.320,390.560,-86.792,-176.175,10.027,148.970
C02546=1138.315,390.847,-86.835,-176.176,10.029,148.971
C02547=1138.311,391.135,-86.879,-176.176,10.032,148.972
C02548=1138.307,391.422,-86.923,-176.176,10.034,148.973
C02549=1138.302,391.669,-86.959,-176.177,10.036,148.973
C02550=1138.299,391.917,-86.997,-176.178,10.039,148.974
C02551=1138.295,392.164,-87.034,-176.179,10.041,148.975
C02552=1138.291,392.411,-87.072,-176.179,10.043,148.976
C02553=1138.289,392.628,-87.104,-176.180,10.045,148.976
C02554=1138.286,392.844,-87.137,-176.180,10.047,148.977
C02555=1138.281,393.061,-87.170,-176.181,10.049,148.978
C02556=1138.265,394.139,-87.330,-176.862,11.324,149.488
C02557=1138.261,394.386,-87.368,-176.861,11.326,149.488
C02558=1138.258,394.633,-87.406,-176.862,11.328,149.489
C02559=1138.254,394.880,-87.442,-176.862,11.329,149.490
C02560=1138.250,395.128,-87.481,-176.862,11.332,149.490
C02561=1138.246,395.374,-87.519,-176.862,11.333,149.491
C02562=1138.242,395.621,-87.555,-176.862,11.336,149.491
C02563=1138.239,395.869,-87.593,-176.863,11.338,149.492
C02564=1138.235,396.115,-87.631,-176.864,11.340,149.492
C02565=1138.231,396.363,-87.668,-176.863,11.342,149.493
C02566=1138.228,396.610,-87.706,-176.864,11.344,149.494
C02567=1138.224,396.857,-87.744,-176.864,11.346,149.494
C02568=1138.220,397.104,-87.781,-176.865,11.348,149.495
C02569=1138.216,397.352,-87.819,-176.865,11.351,149.496
C02570=1138.213,397.598,-87.857,-176.865,11.353,149.496
C02571=1138.209,397.845,-87.894,-176.866,11.355,149.497
C02572=1138.205,398.093,-87.932,-176.866,11.358,149.498
C02573=1138.201,398.340,-87.970,-176.867,11.359,149.498
C02574=1138.198,398.587,-88.008,-176.867,11.362,149.499
C02575=1138.194,398.834,-88.044,-176.868,11.364,149.500
C02576=1138.190,399.081,-88.082,-176.869,11.366,149.501
C02577=1138.187,399.328,-88.120,-176.869,11.369,149.501
C02578=1138.182,399.576,-88.158,-176.870,11.371,149.502
C02579=1138.179,399.823,-88.195,-176.870,11.374,149.503
C02580=1138.175,400.069,-88.233,-176.871,11.376,149.504
C02581=1138.172,400.316,-88.271,-176.872,11.379,149.505
C02582=1138.167,400.564,-88.308,-176.872,11.381,149.505
C02583=1138.164,400.811,-88.346,-176.873,11.383,149.506
C02584=1138.160,401.058,-88.384,-176.874,11.386,149.507
C02585=1138.156,401.306,-88.421,-176.875,11.388,149.508
C02586=1138.152,401.552,-88.459,-176.875,11.391,149.509
C02587=1138.149,401.800,-88.497,-176.876,11.394,149.510
C02588=1138.145,402.046,-88.535,-176.877,11.396,149.511
C02589=1138.142,402.260,-88.567,-176.878,11.398,149.511
C02590=1138.139,402.473,-88.600,-176.879,11.401,149.512
C02591=1138.135,402.686,-88.632,-176.880,11.403,149.513
C02592=1138.132,402.900,-88.664,-176.880,11.406,149.514
C02593=1138.129,403.113,-88.697,-176.881,11.408,149.514
C02594=1138.126,403.327,-88.729,-176.882,11.410,149.515
C02595=1138.122,403.539,-88.762,-176.883,11.412,149.516
C02596=1138.119,403.753,-88.794,-176.883,11.415,149.517
C02597=1138.116,404.000,-88.832,-176.885,11.418,149.518
C02598=1138.112,404.246,-88.870,-176.885,11.421,149.519
C02599=1138.108,404.494,-88.908,-176.887,11.423,149.520
C02600=1138.104,404.741,-88.945,-176.888,11.426,149.521
C02601=1138.101,404.988,-88.983,-176.889,11.429,149.522
C02602=1138.097,405.235,-89.020,-176.890,11.431,149.523
C02603=1138.094,405.482,-89.058,-176.891,11.435,149.524
C02604=1138.089,405.730,-89.096,-176.893,11.437,149.525
C02605=1138.085,405.976,-89.133,-176.894,11.441,149.526
C02606=1138.082,406.224,-89.171,-176.895,11.443,149.527
C02607=1138.078,406.470,-89.209,-176.896,11.447,149.529
C02608=1138.074,406.718,-89.247,-176.898,11.450,149.530
C02609=1138.070,406.965,-89.284,-176.899,11.453,149.531
C02610=1138.067,407.212,-89.322,-176.900,11.456,149.532
C02611=1138.063,407.459,-89.360,-176.901,11.459,149.533
C02612=1138.060,407.707,-89.397,-176.903,11.462,149.534
C02613=1138.055,407.954,-89.435,-176.904,11.465,149.535
C02614=1138.052,408.201,-89.473,-176.906,11.468,149.537
C02615=1138.048,408.447,-89.511,-176.907,11.472,149.538
C02616=1138.045,408.695,-89.549,-176.909,11.475,149.539
C02617=1138.041,408.942,-89.586,-176.910,11.478,149.540
C02618=1138.037,409.189,-89.624,-176.912,11.482,149.542
C02619=1138.033,409.436,-89.662,-176.913,11.485,149.543
C02620=1138.030,409.683,-89.700,-176.916,11.488,149.544
C02621=1138.026,409.931,-89.736,-176.917,11.492,149.545
C02622=1138.022,410.178,-89.775,-176.918,11.496,149.547
C02623=1138.018,410.425,-89.813,-176.920,11.499,149.548
C02624=1138.014,410.671,-89.850,-176.922,11.503,149.549
C02625=1138.011,410.919,-89.888,-176.924,11.506,149.551
C02626=1138.006,411.166,-89.926,-176.925,11.510,149.552
C02627=1138.003,411.413,-89.963,-176.927,11.513,149.554
C02628=1138.000,411.660,-90.001,-176.929,11.517,149.555
C02629=1137.996,411.907,-90.039,-176.930,11.520,149.556
C02630=1137.992,412.154,-90.076,-176.933,11.524,149.558
C02631=1137.988,412.402,-90.114,-176.934,11.528,149.559
C02632=1137.985,412.648,-90.152,-176.937,11.531,149.561
C02633=1137.981,412.896,-90.190,-176.938,11.535,149.562
C02634=1137.978,413.142,-90.227,-176.940,11.539,149.563
C02635=1137.973,413.391,-90.265,-176.942,11.542,149.565
C02636=1137.970,413.637,-90.303,-176.944,11.547,149.567
C02637=1137.966,413.884,-90.341,-176.947,11.550,149.568
C02638=1137.963,414.131,-90.378,-176.949,11.554,149.570
C02639=1137.959,414.379,-90.417,-176.950,11.558,149.571
C02640=1137.955,414.625,-90.453,-176.953,11.562,149.573
C02641=1137.953,414.873,-90.491,-176.955,11.566,149.574
C02642=1137.951,415.119,-90.529,-176.957,11.570,149.576
C02643=1137.950,415.367,-90.566,-176.960,11.574,149.578
C02644=1137.949,415.614,-90.603,-176.961,11.578,149.579
C02645=1137.949,415.826,-90.635,-176.964,11.582,149.581
C02646=1137.950,416.040,-90.667,-176.966,11.585,149.582
C02647=1137.951,416.253,-90.700,-176.967,11.589,149.583
C02648=1137.952,416.466,-90.731,-176.970,11.592,149.585
C02649=1137.954,416.678,-90.763,-176.972,11.596,149.586
C02650=1137.956,416.891,-90.795,-176.974,11.600,149.588
C02651=1137.960,417.103,-90.826,-176.976,11.603,149.589
C02652=1137.962,417.316,-90.858,-176.978,11.607,149.591
C02653=1137.544,417.316,-90.920,-176.971,11.611,149.590
C02654=1137.540,417.104,-90.889,-176.969,11.607,149.589
C02655=1137.537,416.891,-90.857,-176.967,11.604,149.587
C02656=1137.535,416.678,-90.825,-176.964,11.601,149.586
C02657=1137.532,416.465,-90.794,-176.963,11.596,149.584
C02658=1137.531,416.252,-90.762,-176.960,11.593,149.583
C02659=1137.531,416.040,-90.730,-176.959,11.589,149.581
C02660=1137.530,415.827,-90.697,-176.957,11.586,149.580
C02661=1137.530,415.614,-90.666,-176.955,11.582,149.578
C02662=1137.530,415.367,-90.629,-176.952,11.578,149.577
C02663=1137.532,415.120,-90.591,-176.950,11.574,149.575
C02664=1137.533,414.873,-90.554,-176.948,11.570,149.574
C02665=1137.536,414.625,-90.516,-176.946,11.567,149.572
C02666=1137.539,414.378,-90.479,-176.944,11.562,149.570
C02667=1137.543,414.132,-90.440,-176.942,11.558,149.569
C02668=1137.547,413.884,-90.403,-176.940,11.555,149.567
C02669=1137.551,413.637,-90.366,-176.938,11.550,149.566
C02670=1137.554,413.390,-90.328,-176.936,11.546,149.564
C02671=1137.558,413.143,-90.289,-176.933,11.543,149.563
C02672=1137.561,412.896,-90.252,-176.932,11.539,149.561
C02673=1137.566,412.648,-90.215,-176.930,11.535,149.560
C02674=1137.569,412.401,-90.177,-176.928,11.532,149.559
C02675=1137.573,412.154,-90.139,-176.927,11.528,149.557
C02676=1137.576,411.907,-90.101,-176.925,11.523,149.556
C02677=1137.580,411.660,-90.063,-176.923,11.520,149.554
C02678=1137.583,411.413,-90.025,-176.921,11.516,149.553
C02679=1137.588,411.166,-89.988,-176.920,11.513,149.552
C02680=1137.591,410.918,-89.950,-176.918,11.510,149.550
C02681=1137.595,410.672,-89.912,-176.916,11.506,149.549
C02682=1137.598,410.425,-89.874,-176.914,11.503,149.547
C02683=1137.603,410.178,-89.836,-176.913,11.499,149.546
C02684=1137.606,409.930,-89.799,-176.911,11.495,149.545
C02685=1137.610,409.683,-89.761,-176.909,11.492,149.544
C02686=1137.613,409.436,-89.723,-176.908,11.488,149.542
C02687=1137.617,409.189,-89.686,-176.907,11.485,149.541
C02688=1137.621,408.942,-89.647,-176.905,11.482,149.540
C02689=1137.625,408.695,-89.610,-176.904,11.478,149.539
C02690=1137.628,408.447,-89.572,-176.902,11.475,149.537
C02691=1137.632,408.201,-89.535,-176.901,11.472,149.536
C02692=1137.636,407.953,-89.496,-176.899,11.469,149.535
C02693=1137.640,407.707,-89.459,-176.898,11.465,149.534
C02694=1137.643,407.459,-89.421,-176.897,11.462,149.533
C02695=1137.647,407.212,-89.384,-176.895,11.459,149.531
C02696=1137.652,406.965,-89.346,-176.894,11.455,149.530
C02697=1137.655,406.718,-89.308,-176.893,11.453,149.529
C02698=1137.659,406.471,-89.271,-176.891,11.449,149.528
C02699=1137.662,406.224,-89.233,-176.890,11.447,149.527
C02700=1137.666,405.977,-89.195,-176.889,11.443,149.526
C02701=1137.670,405.729,-89.157,-176.887,11.441,149.525
C02702=1137.674,405.483,-89.119,-176.887,11.437,149.524
C02703=1137.677,405.235,-89.082,-176.885,11.435,149.523
C02704=1137.681,404.988,-89.045,-176.884,11.431,149.521
C02705=1137.685,404.741,-89.006,-176.883,11.428,149.520
C02706=1137.689,404.494,-88.968,-176.882,11.426,149.520
C02707=1137.692,404.246,-88.931,-176.881,11.423,149.518
C02708=1137.696,404.000,-88.894,-176.880,11.420,149.518
C02709=1137.699,403.752,-88.856,-176.879,11.417,149.517
C02710=1137.703,403.540,-88.823,-176.878,11.415,149.516
C02711=1137.706,403.326,-88.791,-176.877,11.413,149.515
C02712=1137.709,403.114,-88.758,-176.877,11.410,149.514
C02713=1137.712,402.901,-88.725,-176.876,11.408,149.513
C02714=1137.716,402.688,-88.693,-176.875,11.406,149.513
C02715=1137.719,402.475,-88.661,-176.874,11.404,149.512
C02716=1137.722,402.263,-88.628,-176.874,11.401,149.511
C02717=1137.726,402.049,-88.596,-176.873,11.399,149.510
C02718=1137.729,401.802,-88.558,-176.872,11.396,149.509
C02719=1137.732,401.555,-88.520,-176.871,11.393,149.508
C02720=1137.736,401.309,-88.483,-176.870,11.391,149.508
C02721=1137.741,401.060,-88.445,-176.870,11.388,149.507
C02722=1137.744,400.814,-88.407,-176.869,11.386,149.506
C02723=1137.747,400.567,-88.369,-176.869,11.383,149.505
C02724=1137.752,400.319,-88.332,-176.868,11.381,149.504
C02725=1137.755,400.073,-88.295,-176.868,11.378,149.503
C02726=1137.759,399.825,-88.256,-176.867,11.376,149.503
C02727=1137.763,399.579,-88.219,-176.866,11.373,149.502
C02728=1137.767,399.331,-88.181,-176.865,11.371,149.501
C02729=1137.770,399.084,-88.144,-176.865,11.368,149.500
C02730=1137.774,398.837,-88.106,-176.864,11.366,149.500
C02731=1137.777,398.590,-88.068,-176.864,11.364,149.499
C02732=1137.782,398.342,-88.031,-176.864,11.362,149.498
C02733=1137.785,398.096,-87.993,-176.863,11.359,149.497
C02734=1137.789,397.848,-87.955,-176.863,11.357,149.497
C02735=1137.793,397.601,-87.918,-176.862,11.354,149.496
C02736=1137.796,397.355,-87.881,-176.862,11.352,149.495
C02737=1137.800,397.107,-87.842,-176.861,11.351,149.495
C02738=1137.804,396.860,-87.805,-176.861,11.348,149.494
C02739=1137.808,396.613,-87.767,-176.861,11.346,149.493
C02740=1137.811,396.366,-87.730,-176.861,11.344,149.493
C02741=1137.815,396.119,-87.692,-176.860,11.342,149.492
C02742=1137.819,395.871,-87.655,-176.860,11.339,149.492
C02743=1137.823,395.624,-87.616,-176.860,11.338,149.491
C02744=1137.826,395.377,-87.579,-176.860,11.335,149.490
C02745=1137.831,395.130,-87.542,-176.859,11.333,149.490
C02746=1137.834,394.883,-87.504,-176.860,11.331,149.489
C02747=1137.837,394.636,-87.466,-176.859,11.329,149.489
C02748=1137.841,394.388,-87.429,-176.859,11.328,149.488
C02749=1137.846,394.142,-87.391,-176.859,11.325,149.488
C02750=1137.849,393.894,-87.353,-176.858,11.324,149.487
C02751=1137.853,393.647,-87.316,-176.859,11.321,149.487
C02752=1137.857,393.401,-87.279,-176.859,11.320,149.486
C02753=1137.860,393.153,-87.241,-176.859,11.317,149.485
C02754=1137.864,392.906,-87.204,-176.859,11.316,149.485
C02755=1137.868,392.658,-87.165,-176.859,11.314,149.485
C02756=1137.872,392.412,-87.128,-176.859,11.312,149.484
C02757=1137.875,392.164,-87.091,-176.859,11.310,149.484
C02758=1137.879,391.917,-87.053,-176.859,11.308,149.483
C02759=1137.883,391.671,-87.015,-176.859,11.307,149.483
C02760=1137.886,391.423,-86.978,-176.860,11.305,149.482
C02761=1137.890,391.176,-86.941,-176.859,11.303,149.482
C02762=1137.893,390.928,-86.903,-176.860,11.301,149.482
C02763=1137.898,390.682,-86.865,-176.860,11.300,149.481
C02764=1137.901,390.434,-86.827,-176.860,11.298,149.481
C02765=1137.905,390.187,-86.790,-176.860,11.296,149.480
C02766=1137.910,389.885,-86.745,-176.861,11.294,149.480
C02767=1137.914,389.583,-86.699,-176.861,11.292,149.480
C02768=1137.919,389.281,-86.653,-176.862,11.290,149.479
C02769=1137.923,388.980,-86.607,-176.862,11.288,149.479
C02770=1137.927,388.733,-86.569,-176.862,11.286,149.478
C02771=1137.931,388.486,-86.532,-176.863,11.285,149.478
C02772=1137.934,388.238,-86.494,-176.863,11.283,149.478
C02773=1137.939,387.991,-86.458,-176.863,11.282,149.477
C02774=1137.942,387.744,-86.420,-176.864,11.280,149.477
C02775=1137.946,387.497,-86.382,-176.864,11.279,149.477
C02776=1137.949,387.250,-86.345,-176.865,11.277,149.477
C02777=1137.953,387.003,-86.307,-176.866,11.276,149.476
C02778=1137.957,386.756,-86.270,-176.866,11.274,149.476
C02779=1137.960,386.509,-86.232,-176.867,11.273,149.476
C02780=1137.964,386.261,-86.196,-176.867,11.271,149.476
C02781=1137.967,386.014,-86.158,-176.868,11.270,149.475
C02782=1137.972,385.767,-86.120,-176.869,11.268,149.475
C02783=1137.976,385.520,-86.083,-176.869,11.267,149.475
C02784=1137.980,385.272,-86.045,-176.870,11.265,149.475
C02785=1137.983,385.026,-86.008,-176.870,11.264,149.475
C02786=1137.987,384.778,-85.971,-176.871,11.262,149.474
C02787=1137.991,384.531,-85.933,-176.872,11.261,149.474
C02788=1137.994,384.285,-85.895,-176.873,11.260,149.474
C02789=1137.998,384.037,-85.858,-176.873,11.259,149.474
C02790=1138.002,383.790,-85.821,-176.874,11.257,149.474
C02791=1138.006,383.543,-85.784,-176.875,11.256,149.474
C02792=1138.009,383.295,-85.747,-176.877,11.254,149.474
C02793=1138.013,383.048,-85.709,-176.879,11.252,149.474
C02794=1138.029,381.994,-85.550,-176.190,9.941,148.952
C02795=1138.033,381.784,-85.518,-176.191,9.938,148.951
C02796=1138.036,381.573,-85.487,-176.193,9.935,148.951
C02797=1138.038,381.362,-85.455,-176.194,9.931,148.950
C02798=1138.042,381.115,-85.418,-176.196,9.928,148.950
C02799=1138.046,380.868,-85.381,-176.197,9.925,148.949
C02800=1138.050,380.621,-85.344,-176.199,9.921,148.949
C02801=1138.054,380.373,-85.307,-176.201,9.917,148.948
C02802=1138.058,380.126,-85.270,-176.203,9.914,148.948
C02803=1138.062,379.879,-85.233,-176.204,9.910,148.948
C02804=1138.065,379.632,-85.197,-176.206,9.906,148.947
C02805=1138.069,379.384,-85.159,-176.208,9.903,148.947
C02806=1138.073,379.137,-85.122,-176.210,9.899,148.946
C02807=1138.077,378.890,-85.086,-176.212,9.895,148.946
C02808=1138.081,378.643,-85.049,-176.214,9.892,148.945
C02809=1138.084,378.396,-85.011,-176.215,9.888,148.945
C02810=1138.088,378.149,-84.975,-176.217,9.884,148.944
C02811=1138.092,377.902,-84.938,-176.220,9.880,148.944
C02812=1138.096,377.654,-84.901,-176.222,9.876,148.943
C02813=1138.100,377.407,-84.864,-176.224,9.872,148.943
C02814=1138.103,377.159,-84.827,-176.226,9.869,148.943
C02815=1138.107,376.912,-84.790,-176.228,9.865,148.942
C02816=1138.111,376.665,-84.754,-176.231,9.861,148.942
C02817=1138.115,376.418,-84.717,-176.233,9.857,148.941
C02818=1138.119,376.171,-84.680,-176.235,9.853,148.941
C02819=1138.122,375.923,-84.643,-176.237,9.849,148.940
C02820=1138.126,375.676,-84.606,-176.240,9.845,148.940
C02821=1138.130,375.429,-84.570,-176.242,9.840,148.939
C02822=1138.134,375.181,-84.534,-176.244,9.837,148.939
C02823=1138.138,374.934,-84.497,-176.247,9.832,148.939
C02824=1138.142,374.687,-84.460,-176.249,9.828,148.938
C02825=1138.146,374.440,-84.423,-176.251,9.824,148.938
C02826=1138.149,374.192,-84.387,-176.254,9.820,148.937
C02827=1138.153,373.945,-84.350,-176.256,9.816,148.937
C02828=1138.157,373.698,-84.313,-176.259,9.812,148.936
C02829=1138.160,373.450,-84.278,-176.261,9.808,148.936
C02830=1138.165,373.203,-84.241,-176.263,9.804,148.936
C02831=1138.168,372.956,-84.204,-176.266,9.799,148.935
C02832=1138.172,372.709,-84.168,-176.269,9.795,148.935
C02833=1138.176,372.462,-84.131,-176.271,9.791,148.934
C02834=1138.179,372.214,-84.095,-176.274,9.787,148.934
C02835=1138.183,371.966,-84.058,-176.276,9.782,148.933
C02836=1138.187,371.720,-84.022,-176.278,9.779,148.933
C02837=1138.191,371.472,-83.986,-176.281,9.775,148.933
C02838=1138.194,371.225,-83.949,-176.284,9.770,148.932
C02839=1138.198,370.978,-83.912,-176.286,9.766,148.932
C02840=1138.203,370.730,-83.876,-176.289,9.761,148.931
C02841=1138.206,370.483,-83.840,-176.291,9.757,148.931
C02842=1138.211,370.235,-83.804,-176.294,9.753,148.931
C02843=1138.214,369.988,-83.768,-176.297,9.749,148.930
C02844=1138.218,369.741,-83.731,-176.299,9.744,148.930
C02845=1138.222,369.494,-83.695,-176.302,9.740,148.929
C02846=1138.226,369.246,-83.658,-176.305,9.736,148.929
C02847=1138.229,368.999,-83.623,-176.307,9.731,148.929
C02848=1138.234,368.752,-83.586,-176.310,9.727,148.928
C02849=1138.237,368.504,-83.550,-176.312,9.723,148.928
C02850=1138.241,368.257,-83.514,-176.315,9.719,148.927
C02851=1138.245,368.010,-83.478,-176.318,9.714,148.927
C02852=1138.248,367.763,-83.442,-176.320,9.710,148.926
C02853=1138.253,367.515,-83.406,-176.323,9.706,148.926
C02854=1138.256,367.267,-83.370,-176.326,9.701,148.926
C02855=1138.261,367.020,-83.333,-176.328,9.697,148.925
C02856=1138.264,366.773,-83.298,-176.331,9.693,148.925
C02857=1138.268,366.526,-83.261,-176.334,9.689,148.924
C02858=1138.272,366.278,-83.225,-176.336,9.684,148.924
C02859=1138.276,366.030,-83.190,-176.339,9.680,148.924
C02860=1138.279,365.784,-83.153,-176.341,9.675,148.923
C02861=1138.283,365.536,-83.117,-176.344,9.671,148.923
C02862=1138.288,365.252,-83.076,-176.347,9.666,148.922
C02863=1138.292,364.968,-83.035,-176.351,9.661,148.922
C02864=1138.296,364.684,-82.994,-176.353,9.657,148.921
C02865=1138.301,364.401,-82.953,-176.356,9.651,148.921
C02866=1138.305,364.153,-82.917,-176.359,9.647,148.921
C02867=1138.309,363.905,-82.881,-176.362,9.643,148.920
C02868=1138.312,363.658,-82.846,-176.364,9.639,148.920
C02869=1138.316,363.410,-82.810,-176.367,9.634,148.919
C02870=1138.320,363.163,-82.773,-176.370,9.630,148.919
C02871=1138.324,362.916,-82.738,-176.372,9.626,148.918
C02872=1138.328,362.669,-82.702,-176.375,9.621,148.918
C02873=1138.332,362.421,-82.667,-176.378,9.617,148.918
C02874=1138.335,362.174,-82.631,-176.380,9.614,148.917
C02875=1138.340,361.926,-82.595,-176.382,9.609,148.917
C02876=1138.343,361.678,-82.560,-176.385,9.605,148.916
C02877=1138.347,361.431,-82.524,-176.388,9.601,148.916
C02878=1138.351,361.184,-82.489,-176.390,9.596,148.916
C02879=1138.355,360.937,-82.453,-176.393,9.592,148.915
C02880=1138.359,360.689,-82.418,-176.395,9.588,148.915
C02881=1138.362,360.442,-82.382,-176.398,9.584,148.915
C02882=1138.367,360.194,-82.346,-176.401,9.579,148.914
C02883=1138.370,359.946,-82.311,-176.402,9.576,148.914
C02884=1138.375,359.700,-82.275,-176.405,9.572,148.913
C02885=1138.378,359.452,-82.240,-176.408,9.567,148.913
C02886=1138.382,359.205,-82.204,-176.410,9.563,148.913
C02887=1138.386,358.957,-82.169,-176.413,9.559,148.912
C02888=1138.390,358.709,-82.134,-176.416,9.554,148.912
C02889=1138.394,358.462,-82.099,-176.418,9.551,148.911
C02890=1138.398,358.215,-82.063,-176.420,9.546,148.911
C02891=1138.401,357.967,-82.028,-176.423,9.542,148.911
C02892=1138.405,357.720,-81.992,-176.426,9.538,148.910
C02893=1138.409,357.473,-81.957,-176.428,9.534,148.910
C02894=1138.413,357.225,-81.922,-176.431,9.530,148.910
C02895=1138.417,356.977,-81.887,-176.433,9.526,148.909
C02896=1138.420,356.730,-81.851,-176.436,9.522,148.909
C02897=1138.425,356.483,-81.816,-176.439,9.518,148.908
C02898=1138.429,356.235,-81.781,-176.441,9.513,148.908
C02899=1138.432,355.987,-81.745,-176.443,9.510,148.908
C02900=1138.437,355.740,-81.710,-176.446,9.506,148.907
C02901=1138.441,355.492,-81.675,-176.448,9.501,148.907
C02902=1138.444,355.245,-81.640,-176.451,9.497,148.906
C02903=1138.448,354.997,-81.604,-176.453,9.493,148.906
C02904=1138.452,354.750,-81.570,-176.456,9.489,148.906
C02905=1138.456,354.502,-81.534,-176.458,9.485,148.905
C02906=1138.460,354.254,-81.499,-176.461,9.481,148.905
C02907=1138.464,354.007,-81.464,-176.463,9.477,148.905
C02908=1138.468,353.760,-81.429,-176.466,9.473,148.904
C02909=1138.471,353.512,-81.394,-176.469,9.469,148.904
C02910=1138.475,353.265,-81.359,-176.471,9.464,148.903
C02911=1138.479,353.017,-81.324,-176.473,9.461,148.903
C02912=1138.483,352.770,-81.289,-176.476,9.457,148.903
C02913=1138.488,352.522,-81.254,-176.479,9.452,148.902
C02914=1138.491,352.275,-81.219,-176.481,9.448,148.902
C02915=1138.496,352.027,-81.184,-176.483,9.445,148.902
C02916=1138.499,351.780,-81.150,-176.486,9.440,148.901
C02917=1138.503,351.532,-81.115,-176.489,9.436,148.901
C02918=1138.507,351.285,-81.080,-176.491,9.432,148.901
C02919=1138.511,351.037,-81.045,-176.494,9.428,148.900
C02920=1138.516,350.790,-81.010,-176.496,9.424,148.900
C02921=1138.519,350.542,-80.976,-176.499,9.420,148.899
C02922=1138.522,350.294,-80.940,-176.501,9.416,148.899
C02923=1138.527,350.047,-80.906,-176.504,9.412,148.899
C02924=1138.531,349.799,-80.871,-176.507,9.408,148.899
C02925=1138.535,349.552,-80.837,-176.509,9.404,148.898
C02926=1138.539,349.304,-80.802,-176.511,9.400,148.898
C02927=1138.543,349.057,-80.767,-176.514,9.396,148.897
C02928=1138.547,348.809,-80.732,-176.516,9.392,148.897
C02929=1138.551,348.562,-80.698,-176.519,9.388,148.897
C02930=1138.555,348.314,-80.663,-176.521,9.384,148.896
C02931=1138.559,348.066,-80.628,-176.524,9.380,148.896
C02932=1138.562,347.819,-80.594,-176.527,9.376,148.896
C02933=1138.566,347.571,-80.559,-176.529,9.372,148.895
C02934=1138.571,347.324,-80.524,-176.532,9.368,148.895
C02935=1138.574,347.076,-80.490,-176.534,9.364,148.895
C02936=1138.578,346.829,-80.456,-176.536,9.360,148.894
C02937=1138.582,346.581,-80.421,-176.539,9.356,148.894
C02938=1138.586,346.334,-80.387,-176.542,9.352,148.894
C02939=1138.591,346.086,-80.352,-176.545,9.348,148.893
C02940=1138.594,345.838,-80.318,-176.547,9.344,148.893
C02941=1138.599,345.591,-80.284,-176.550,9.340,148.893
C02942=1138.603,345.343,-80.249,-176.552,9.336,148.892
C02943=1138.606,345.096,-80.215,-176.554,9.332,148.892
C02944=1138.610,344.848,-80.180,-176.557,9.328,148.892
C02945=1138.614,344.600,-80.146,-176.560,9.324,148.891
C02946=1138.618,344.352,-80.111,-176.562,9.320,148.891
C02947=1138.622,344.105,-80.078,-176.565,9.316,148.891
C02948=1138.626,343.857,-80.043,-176.567,9.312,148.890
C02949=1138.630,343.610,-80.009,-176.570,9.309,148.890
C02950=1138.634,343.363,-79.974,-176.572,9.304,148.890
C02951=1138.638,343.115,-79.940,-176.575,9.300,148.889
C02952=1138.642,342.867,-79.906,-176.577,9.297,148.889
C02953=1138.645,342.620,-79.871,-176.580,9.293,148.889
C02954=1138.650,342.372,-79.837,-176.583,9.288,148.888
C02955=1138.654,342.125,-79.803,-176.585,9.285,148.888
C02956=1138.658,341.876,-79.769,-176.588,9.281,148.888
C02957=1138.662,341.629,-79.735,-176.590,9.276,148.887
C02958=1138.666,341.382,-79.701,-176.593,9.273,148.887
C02959=1138.670,341.134,-79.666,-176.595,9.269,148.887
C02960=1138.675,340.886,-79.633,-176.598,9.265,148.887
C02961=1138.678,340.638,-79.598,-176.600,9.261,148.886
C02962=1138.682,340.391,-79.565,-176.603,9.257,148.886
C02963=1138.686,340.144,-79.530,-176.606,9.253,148.886
C02964=1138.690,339.895,-79.497,-176.608,9.250,148.885
C02965=1138.694,339.648,-79.462,-176.611,9.245,148.885
C02966=1138.699,339.367,-79.424,-176.614,9.241,148.885
C02967=1138.703,339.087,-79.386,-176.617,9.236,148.884
C02968=1138.708,338.806,-79.347,-176.620,9.232,148.884
C02969=1138.712,338.525,-79.308,-176.622,9.228,148.884
C02970=1138.716,338.277,-79.274,-176.625,9.224,148.883
C02971=1138.721,338.030,-79.241,-176.627,9.220,148.883
C02972=1138.724,337.783,-79.207,-176.630,9.216,148.883
C02973=1138.728,337.534,-79.173,-176.633,9.212,148.882
C02974=1138.733,337.287,-79.139,-176.635,9.209,148.882
C02975=1138.737,337.039,-79.106,-176.638,9.204,148.882
C02976=1138.740,336.791,-79.071,-176.641,9.200,148.882
C02977=1138.744,336.544,-79.038,-176.643,9.197,148.881
C02978=1138.749,336.296,-79.004,-176.645,9.193,148.881
C02979=1138.753,336.048,-78.971,-176.648,9.189,148.881
C02980=1138.756,335.801,-78.936,-176.651,9.185,148.880
C02981=1138.760,335.553,-78.903,-176.653,9.181,148.880
C02982=1138.765,335.305,-78.869,-176.656,9.178,148.880
C02983=1138.769,335.058,-78.836,-176.658,9.173,148.880
C02984=1138.772,334.810,-78.801,-176.661,9.169,148.879
C02985=1138.776,334.562,-78.768,-176.663,9.166,148.879
C02986=1138.780,334.314,-78.735,-176.666,9.162,148.879
C02987=1138.784,334.067,-78.701,-176.669,9.159,148.879
C02988=1138.788,333.819,-78.667,-176.671,9.154,148.878
C02989=1138.793,333.571,-78.634,-176.674,9.150,148.878
C02990=1138.796,333.324,-78.600,-176.676,9.147,148.878
C02991=1138.801,333.076,-78.567,-176.679,9.143,148.877
C02992=1138.805,332.828,-78.534,-176.681,9.139,148.877
C02993=1138.809,332.581,-78.500,-176.684,9.135,148.877
C02994=1138.812,332.333,-78.466,-176.687,9.131,148.877
C02995=1138.816,332.085,-78.433,-176.689,9.128,148.876
C02996=1138.820,331.837,-78.400,-176.692,9.123,148.876
C02997=1138.824,331.590,-78.366,-176.694,9.120,148.876
C02998=1138.828,331.342,-78.333,-176.697,9.116,148.876
C02999=1138.833,331.094,-78.299,-176.700,9.112,148.875
C03000=1138.837,330.846,-78.266,-176.702,9.108,148.875
C03001=1138.841,330.598,-78.233,-176.705,9.104,148.875
C03002=1138.845,330.350,-78.200,-176.707,9.101,148.874
C03003=1138.849,330.103,-78.166,-176.710,9.097,148.874
C03004=1138.853,329.856,-78.132,-176.712,9.093,148.874
C03005=1138.857,329.608,-78.099,-176.715,9.089,148.874
C03006=1138.861,329.360,-78.066,-176.718,9.085,148.873
C03007=1138.865,329.112,-78.033,-176.720,9.082,148.873
C03008=1138.870,328.865,-78.000,-176.723,9.078,148.873
C03009=1138.873,328.616,-77.966,-176.725,9.074,148.873
C03010=1138.876,328.369,-77.934,-176.728,9.070,148.872
C03011=1138.881,328.121,-77.901,-176.730,9.067,148.872
C03012=1138.885,327.873,-77.867,-176.733,9.063,148.872
C03013=1138.889,327.626,-77.834,-176.736,9.059,148.872
C03014=1138.893,327.378,-77.801,-176.739,9.056,148.871
C03015=1138.897,327.130,-77.768,-176.741,9.051,148.871
C03016=1138.901,326.882,-77.735,-176.744,9.048,148.871
C03017=1138.905,326.635,-77.702,-176.746,9.044,148.871
C03018=1138.910,326.387,-77.669,-176.749,9.041,148.870
C03019=1138.914,326.139,-77.636,-176.752,9.037,148.870
C03020=1138.917,325.891,-77.604,-176.754,9.033,148.870
C03021=1138.922,325.644,-77.570,-176.757,9.029,148.870
C03022=1138.926,325.396,-77.537,-176.759,9.025,148.869
C03023=1138.930,325.148,-77.504,-176.762,9.022,148.869
C03024=1138.934,324.900,-77.471,-176.765,9.018,148.869
C03025=1138.938,324.652,-77.438,-176.767,9.014,148.869
C03026=1138.942,324.405,-77.406,-176.770,9.010,148.868
C03027=1138.946,324.157,-77.373,-176.772,9.007,148.868
C03028=1138.950,323.909,-77.340,-176.775,9.003,148.868
C03029=1138.955,323.661,-77.307,-176.778,9.000,148.868
C03030=1138.958,323.413,-77.275,-176.781,8.996,148.868
C03031=1138.962,323.166,-77.241,-176.782,8.992,148.867
C03032=1138.966,322.918,-77.208,-176.785,8.988,148.867
C03033=1138.971,322.670,-77.176,-176.788,8.985,148.867
C03034=1138.974,322.422,-77.143,-176.791,8.981,148.867
C03035=1138.978,322.174,-77.110,-176.794,8.977,148.866
C03036=1138.983,321.926,-77.078,-176.796,8.973,148.866
C03037=1138.986,321.679,-77.045,-176.799,8.969,148.866
C03038=1138.990,321.430,-77.013,-176.801,8.966,148.866
C03039=1138.995,321.183,-76.980,-176.804,8.962,148.866
C03040=1138.998,320.935,-76.947,-176.807,8.959,148.865
C03041=1139.003,320.687,-76.915,-176.809,8.955,148.865
C03042=1139.007,320.440,-76.882,-176.812,8.951,148.865
C03043=1139.011,320.192,-76.850,-176.815,8.947,148.865
C03044=1139.015,319.944,-76.817,-176.817,8.944,148.865
C03045=1139.019,319.696,-76.784,-176.820,8.940,148.864
C03046=1139.023,319.448,-76.752,-176.822,8.937,148.864
C03047=1139.027,319.200,-76.719,-176.825,8.933,148.864
C03048=1139.031,318.952,-76.687,-176.828,8.929,148.864
C03049=1139.035,318.704,-76.654,-176.831,8.925,148.863
C03050=1139.039,318.457,-76.622,-176.833,8.922,148.863
C03051=1139.044,318.209,-76.590,-176.836,8.918,148.863
C03052=1139.048,317.961,-76.557,-176.838,8.915,148.863
C03053=1139.051,317.713,-76.525,-176.841,8.911,148.863
C03054=1139.056,317.465,-76.492,-176.843,8.907,148.862
C03055=1139.060,317.217,-76.460,-176.846,8.903,148.862
C03056=1139.064,316.969,-76.427,-176.849,8.900,148.862
C03057=1139.068,316.722,-76.396,-176.852,8.896,148.862
C03058=1139.073,316.473,-76.363,-176.854,8.893,148.862
C03059=1139.076,316.226,-76.331,-176.857,8.889,148.861
C03060=1139.080,315.978,-76.298,-176.859,8.885,148.861
C03061=1139.084,315.730,-76.266,-176.862,8.881,148.861
C03062=1139.089,315.483,-76.234,-176.865,8.878,148.861
C03063=1139.092,315.235,-76.202,-176.867,8.875,148.861
C03064=1139.097,314.986,-76.169,-176.870,8.871,148.860
C03065=1139.101,314.738,-76.138,-176.872,8.867,148.860
C03066=1139.104,314.490,-76.106,-176.875,8.863,148.860
C03067=1139.109,314.243,-76.073,-176.877,8.860,148.860
C03068=1139.113,313.995,-76.041,-176.880,8.856,148.860
C03069=1139.117,313.747,-76.009,-176.883,8.853,148.859
C03070=1139.122,313.469,-75.973,-176.886,8.849,148.859
C03071=1139.127,313.191,-75.937,-176.889,8.845,148.859
C03072=1139.130,312.913,-75.901,-176.891,8.841,148.859
C03073=1139.136,312.635,-75.865,-176.895,8.837,148.859
C03074=1139.140,312.387,-75.834,-176.898,8.833,148.859
C03075=1139.143,312.140,-75.801,-176.900,8.829,148.858
C03076=1139.148,311.892,-75.769,-176.903,8.825,148.858
C03077=1139.152,311.644,-75.737,-176.905,8.822,148.858
C03078=1139.156,311.396,-75.706,-176.908,8.818,148.858
C03079=1139.160,311.148,-75.673,-176.911,8.815,148.858
C03080=1139.164,310.900,-75.641,-176.913,8.812,148.857
C03081=1139.168,310.652,-75.610,-176.916,8.807,148.857
C03082=1139.173,310.403,-75.578,-176.919,8.805,148.857
C03083=1139.177,310.155,-75.546,-176.922,8.800,148.857
C03084=1139.181,309.908,-75.515,-176.924,8.797,148.857
C03085=1139.185,309.660,-75.483,-176.927,8.793,148.857
C03086=1139.189,309.412,-75.450,-176.929,8.790,148.856
C03087=1139.194,309.164,-75.419,-176.932,8.786,148.856
C03088=1139.197,308.916,-75.387,-176.934,8.783,148.856
C03089=1139.201,308.668,-75.355,-176.937,8.780,148.856
C03090=1139.206,308.421,-75.323,-176.940,8.776,148.856
C03091=1139.210,308.172,-75.292,-176.943,8.772,148.856
C03092=1139.214,307.925,-75.261,-176.945,8.768,148.855
C03093=1139.218,307.677,-75.229,-176.948,8.765,148.855
C03094=1139.222,307.429,-75.197,-176.950,8.762,148.855
C03095=1139.227,307.180,-75.166,-176.954,8.758,148.855
C03096=1139.231,306.932,-75.134,-176.956,8.755,148.855
C03097=1139.235,306.685,-75.102,-176.959,8.751,148.855
C03098=1139.239,306.437,-75.070,-176.961,8.747,148.854
C03099=1139.243,306.188,-75.039,-176.964,8.743,148.854
C03100=1139.247,305.941,-75.008,-176.967,8.740,148.854
C03101=1139.251,305.693,-74.976,-176.969,8.737,148.854
C03102=1139.255,305.445,-74.945,-176.972,8.733,148.854
C03103=1139.260,305.197,-74.913,-176.974,8.730,148.854
C03104=1139.264,304.949,-74.881,-176.977,8.726,148.853
C03105=1139.268,304.701,-74.850,-176.980,8.723,148.854
C03106=1139.273,304.453,-74.819,-176.983,8.720,148.853
C03107=1139.277,304.205,-74.787,-176.985,8.715,148.853
C03108=1139.281,303.957,-74.756,-176.988,8.712,148.853
C03109=1139.285,303.709,-74.724,-176.991,8.708,148.853
C03110=1139.289,303.461,-74.693,-176.993,8.705,148.853
C03111=1139.293,303.213,-74.662,-176.996,8.702,148.853
C03112=1139.297,302.965,-74.631,-176.999,8.698,148.852
C03113=1139.301,302.717,-74.599,-177.001,8.695,148.852
C03114=1139.306,302.469,-74.568,-177.004,8.691,148.852
C03115=1139.309,302.221,-74.536,-177.007,8.688,148.852
C03116=1139.314,301.973,-74.506,-177.009,8.684,148.852
C03117=1139.318,301.725,-74.474,-177.013,8.681,148.852
C03118=1139.322,301.477,-74.443,-177.015,8.677,148.852
C03119=1139.326,301.229,-74.412,-177.017,8.674,148.852
C03120=1139.331,300.981,-74.380,-177.020,8.670,148.851
C03121=1139.335,300.733,-74.349,-177.023,8.667,148.851
C03122=1139.339,300.485,-74.318,-177.026,8.663,148.851
C03123=1139.343,300.237,-74.287,-177.028,8.660,148.851
C03124=1139.348,299.989,-74.256,-177.031,8.657,148.851
C03125=1139.351,299.740,-74.225,-177.034,8.653,148.851
C03126=1139.355,299.493,-74.194,-177.036,8.649,148.851
C03127=1139.360,299.245,-74.163,-177.039,8.646,148.850
C03128=1139.364,298.996,-74.132,-177.042,8.642,148.850
C03129=1139.368,298.749,-74.100,-177.044,8.639,148.850
C03130=1139.372,298.500,-74.069,-177.047,8.636,148.850
C03131=1139.377,298.252,-74.039,-177.050,8.632,148.850
C03132=1139.381,298.005,-74.008,-177.052,8.629,148.850
C03133=1139.384,297.757,-73.977,-177.055,8.626,148.850
C03134=1139.389,297.509,-73.946,-177.058,8.622,148.850
C03135=1139.393,297.260,-73.915,-177.060,8.619,148.850
C03136=1139.398,297.012,-73.884,-177.063,8.615,148.849
C03137=1139.402,296.764,-73.854,-177.066,8.612,148.849
C03138=1139.406,296.516,-73.823,-177.068,8.608,148.849
C03139=1139.410,296.268,-73.791,-177.071,8.604,148.849
C03140=1139.414,296.020,-73.760,-177.074,8.601,148.849
C03141=1139.418,295.772,-73.730,-177.076,8.598,148.849
C03142=1139.422,295.524,-73.699,-177.079,8.594,148.849
C03143=1139.427,295.276,-73.668,-177.082,8.591,148.849
C03144=1139.431,295.028,-73.637,-177.085,8.588,148.849
C03145=1139.435,294.780,-73.607,-177.088,8.584,148.849
C03146=1139.439,294.532,-73.576,-177.090,8.581,148.848
C03147=1139.443,294.283,-73.545,-177.093,8.578,148.848
C03148=1139.447,294.036,-73.515,-177.096,8.574,148.848
C03149=1139.452,293.788,-73.484,-177.098,8.571,148.848
C03150=1139.456,293.539,-73.453,-177.101,8.567,148.848
C03151=1139.460,293.291,-73.423,-177.104,8.564,148.848
C03152=1139.464,293.043,-73.392,-177.106,8.560,148.848
C03153=1139.468,292.795,-73.361,-177.109,8.557,148.848
C03154=1139.472,292.547,-73.331,-177.111,8.554,148.848
C03155=1139.477,292.299,-73.300,-177.114,8.550,148.847
C03156=1139.481,292.051,-73.271,-177.117,8.547,148.847
C03157=1139.485,291.802,-73.239,-177.120,8.544,148.847
C03158=1139.490,291.554,-73.209,-177.123,8.540,148.847
C03159=1139.494,291.307,-73.179,-177.125,8.537,148.847
C03160=1139.498,291.059,-73.148,-177.128,8.534,148.847
C03161=1139.502,290.810,-73.117,-177.131,8.530,148.847
C03162=1139.506,290.562,-73.087,-177.133,8.527,148.847
C03163=1139.510,290.314,-73.057,-177.136,8.524,148.847
C03164=1139.515,290.066,-73.026,-177.139,8.520,148.847
C03165=1139.519,289.819,-72.996,-177.142,8.517,148.847
C03166=1139.523,289.570,-72.965,-177.144,8.514,148.846
C03167=1139.527,289.322,-72.935,-177.147,8.511,148.846
C03168=1139.532,289.074,-72.905,-177.150,8.507,148.846
C03169=1139.536,288.826,-72.875,-177.153,8.504,148.846
C03170=1139.540,288.577,-72.845,-177.155,8.500,148.846
C03171=1139.544,288.329,-72.814,-177.158,8.496,148.846
C03172=1139.548,288.081,-72.783,-177.161,8.493,148.846
C03173=1139.552,287.833,-72.754,-177.163,8.490,148.846
C03174=1139.557,287.557,-72.719,-177.166,8.486,148.846
C03175=1139.562,287.282,-72.686,-177.169,8.482,148.846
C03176=1139.566,287.006,-72.653,-177.172,8.479,148.846
C03177=1139.572,286.731,-72.619,-177.175,8.476,148.846
C03178=1139.575,286.482,-72.589,-177.178,8.472,148.846
C03179=1139.580,286.234,-72.559,-177.181,8.469,148.846
C03180=1139.584,285.986,-72.529,-177.184,8.465,148.845
C03181=1139.588,285.738,-72.499,-177.186,8.462,148.845
C03182=1139.593,285.490,-72.469,-177.189,8.458,148.845
C03183=1139.597,285.242,-72.439,-177.192,8.455,148.845
C03184=1139.601,284.994,-72.409,-177.194,8.452,148.845
C03185=1139.605,284.746,-72.379,-177.197,8.449,148.845
C03186=1139.610,284.498,-72.349,-177.200,8.445,148.845
C03187=1139.613,284.249,-72.319,-177.203,8.442,148.845
C03188=1139.618,284.001,-72.289,-177.205,8.439,148.845
C03189=1139.622,283.753,-72.258,-177.208,8.436,148.845
C03190=1139.626,283.505,-72.229,-177.211,8.432,148.845
C03191=1139.631,283.256,-72.199,-177.214,8.429,148.845
C03192=1139.635,283.008,-72.169,-177.216,8.426,148.845
C03193=1139.639,282.760,-72.139,-177.219,8.423,148.845
C03194=1139.643,282.512,-72.110,-177.222,8.419,148.844
C03195=1139.648,282.264,-72.079,-177.225,8.416,148.844
C03196=1139.652,282.016,-72.050,-177.227,8.413,148.844
C03197=1139.656,281.767,-72.020,-177.230,8.410,148.844
C03198=1139.660,281.520,-71.990,-177.233,8.406,148.844
C03199=1139.665,281.271,-71.960,-177.235,8.403,148.844
C03200=1139.669,281.023,-71.931,-177.238,8.400,148.844
C03201=1139.673,280.775,-71.901,-177.241,8.396,148.844
C03202=1139.677,280.526,-71.872,-177.244,8.393,148.844
C03203=1139.681,280.279,-71.841,-177.246,8.389,148.844
C03204=1139.686,280.030,-71.811,-177.249,8.387,148.844
C03205=1139.690,279.782,-71.782,-177.252,8.384,148.844
C03206=1139.695,279.534,-71.752,-177.255,8.380,148.844
C03207=1139.699,279.285,-71.723,-177.258,8.377,148.844
C03208=1139.703,279.037,-71.694,-177.260,8.373,148.844
C03209=1139.707,278.789,-71.663,-177.263,8.370,148.844
C03210=1139.711,278.541,-71.634,-177.265,8.367,148.844
C03211=1139.715,278.293,-71.604,-177.268,8.363,148.844
C03212=1139.720,278.044,-71.574,-177.271,8.361,148.844
C03213=1139.724,277.796,-71.545,-177.273,8.357,148.844
C03214=1139.728,277.548,-71.516,-177.276,8.354,148.844
C03215=1139.733,277.300,-71.486,-177.279,8.351,148.844
C03216=1139.737,277.051,-71.457,-177.282,8.347,148.843
C03217=1139.741,276.803,-71.427,-177.285,8.344,148.843
C03218=1139.745,276.555,-71.398,-177.287,8.341,148.843
C03219=1139.750,276.307,-71.369,-177.290,8.338,148.843
C03220=1139.754,276.059,-71.339,-177.293,8.335,148.843
C03221=1139.758,275.811,-71.310,-177.296,8.331,148.843
C03222=1139.762,275.562,-71.280,-177.298,8.328,148.843
C03223=1139.767,275.314,-71.251,-177.301,8.325,148.843
C03224=1139.771,275.066,-71.221,-177.304,8.322,148.843
C03225=1139.775,274.818,-71.192,-177.307,8.318,148.843
C03226=1139.779,274.569,-71.162,-177.309,8.315,148.843
C03227=1139.784,274.320,-71.134,-177.312,8.312,148.843
C03228=1139.788,274.073,-71.105,-177.315,8.309,148.843
C03229=1139.793,273.825,-71.075,-177.317,8.306,148.843
C03230=1139.797,273.576,-71.046,-177.320,8.303,148.843
C03231=1139.801,273.328,-71.016,-177.323,8.299,148.843
C03232=1139.804,273.080,-70.987,-177.326,8.296,148.843
C03233=1139.809,272.831,-70.959,-177.328,8.293,148.843
C03234=1139.814,272.584,-70.930,-177.331,8.290,148.843
C03235=1139.818,272.335,-70.900,-177.334,8.287,148.843
C03236=1139.822,272.087,-70.871,-177.337,8.283,148.843
C03237=1139.827,271.838,-70.842,-177.340,8.280,148.843
C03238=1139.831,271.590,-70.812,-177.342,8.277,148.843
C03239=1139.835,271.342,-70.783,-177.345,8.274,148.843
C03240=1139.839,271.094,-70.755,-177.348,8.271,148.843
C03241=1139.843,270.846,-70.726,-177.350,8.268,148.843
C03242=1139.848,270.597,-70.696,-177.353,8.264,148.843
C03243=1139.852,270.348,-70.668,-177.356,8.261,148.843
C03244=1139.857,270.101,-70.639,-177.359,8.258,148.843
C03245=1139.860,269.853,-70.610,-177.361,8.255,148.843
C03246=1139.865,269.604,-70.581,-177.364,8.252,148.843
C03247=1139.869,269.356,-70.551,-177.367,8.249,148.843
C03248=1139.874,269.108,-70.523,-177.370,8.245,148.843
C03249=1139.878,268.859,-70.494,-177.373,8.242,148.843
C03250=1139.882,268.611,-70.466,-177.375,8.239,148.843
C03251=1139.886,268.362,-70.436,-177.378,8.236,148.843
C03252=1139.891,268.114,-70.408,-177.381,8.233,148.843
C03253=1139.896,267.866,-70.378,-177.383,8.230,148.843
C03254=1139.899,267.617,-70.350,-177.387,8.227,148.843
C03255=1139.903,267.369,-70.321,-177.389,8.223,148.843
C03256=1139.909,267.121,-70.292,-177.392,8.220,148.843
C03257=1139.912,266.873,-70.263,-177.395,8.217,148.843
C03258=1139.916,266.624,-70.235,-177.397,8.215,148.843
C03259=1139.921,266.377,-70.206,-177.400,8.211,148.843
C03260=1139.925,266.128,-70.177,-177.403,8.208,148.843
C03261=1139.929,265.879,-70.149,-177.406,8.205,148.843
C03262=1139.934,265.631,-70.120,-177.409,8.202,148.843
C03263=1139.938,265.383,-70.091,-177.411,8.198,148.843
C03264=1139.942,265.135,-70.062,-177.414,8.196,148.843
C03265=1139.947,264.886,-70.034,-177.417,8.193,148.843
C03266=1139.951,264.638,-70.006,-177.419,8.190,148.843
C03267=1139.956,264.389,-69.977,-177.422,8.186,148.843
C03268=1139.960,264.142,-69.948,-177.425,8.183,148.843
C03269=1139.964,263.893,-69.920,-177.428,8.180,148.843
C03270=1139.969,263.645,-69.891,-177.431,8.177,148.843
C03271=1139.973,263.397,-69.862,-177.433,8.174,148.843
C03272=1139.977,263.148,-69.834,-177.436,8.171,148.843
C03273=1139.981,262.900,-69.806,-177.439,8.168,148.843
C03274=1139.986,262.651,-69.777,-177.441,8.165,148.843
C03275=1139.990,262.403,-69.749,-177.444,8.162,148.843
C03276=1139.994,262.155,-69.720,-177.447,8.159,148.843
C03277=1139.998,261.906,-69.692,-177.450,8.155,148.843
C03278=1140.004,261.633,-69.660,-177.453,8.152,148.843
C03279=1140.008,261.359,-69.630,-177.456,8.148,148.843
C03280=1140.013,261.085,-69.598,-177.459,8.145,148.843
C03281=1140.017,260.812,-69.567,-177.462,8.142,148.843
C03282=1140.023,260.564,-69.538,-177.465,8.139,148.843
C03283=1140.026,260.316,-69.510,-177.467,8.135,148.843
C03284=1140.031,260.067,-69.481,-177.470,8.132,148.843
C03285=1140.035,259.819,-69.454,-177.473,8.130,148.843
C03286=1140.039,259.570,-69.426,-177.476,8.127,148.843
C03287=1140.044,259.322,-69.397,-177.479,8.124,148.843
C03288=1140.048,259.073,-69.369,-177.481,8.120,148.843
C03289=1140.053,258.825,-69.341,-177.484,8.118,148.843
C03290=1140.057,258.577,-69.312,-177.487,8.114,148.843
C03291=1140.061,258.329,-69.285,-177.490,8.111,148.843
C03292=1140.065,258.080,-69.256,-177.493,8.108,148.843
C03293=1140.070,257.832,-69.228,-177.495,8.105,148.843
C03294=1140.074,257.583,-69.199,-177.498,8.102,148.843
C03295=1140.079,257.335,-69.172,-177.501,8.099,148.843
C03296=1140.082,257.087,-69.144,-177.503,8.096,148.843
C03297=1140.088,256.838,-69.116,-177.506,8.093,148.843
C03298=1140.091,256.589,-69.088,-177.509,8.090,148.843
C03299=1140.096,256.341,-69.060,-177.512,8.087,148.843
C03300=1140.100,256.093,-69.032,-177.514,8.084,148.843
C03301=1140.105,255.845,-69.003,-177.517,8.081,148.843
C03302=1140.109,255.597,-68.976,-177.520,8.078,148.843
C03303=1140.113,255.348,-68.948,-177.523,8.074,148.844
C03304=1140.118,255.099,-68.920,-177.526,8.071,148.844
C03305=1140.122,254.851,-68.892,-177.529,8.069,148.844
C03306=1140.126,254.603,-68.864,-177.531,8.066,148.844
C03307=1140.130,254.354,-68.836,-177.534,8.063,148.844
C03308=1140.135,254.106,-68.808,-177.537,8.059,148.844
C03309=1140.140,253.858,-68.780,-177.539,8.057,148.844
C03310=1140.143,253.609,-68.752,-177.542,8.054,148.844
C03311=1140.148,253.361,-68.725,-177.545,8.051,148.844
C03312=1140.152,253.112,-68.697,-177.548,8.048,148.844
C03313=1140.157,252.864,-68.669,-177.551,8.045,148.844
C03314=1140.162,252.615,-68.642,-177.553,8.042,148.844
C03315=1140.165,252.367,-68.613,-177.556,8.039,148.844
C03316=1140.170,252.119,-68.586,-177.559,8.036,148.844
C03317=1140.174,251.870,-68.558,-177.561,8.033,148.844
C03318=1140.178,251.622,-68.530,-177.564,8.030,148.844
C03319=1140.183,251.373,-68.503,-177.567,8.027,148.844
C03320=1140.187,251.124,-68.475,-177.570,8.024,148.844
C03321=1140.192,250.877,-68.447,-177.573,8.021,148.844
C03322=1140.196,250.628,-68.420,-177.576,8.017,148.844
C03323=1140.200,250.379,-68.392,-177.579,8.015,148.844
C03324=1140.205,250.131,-68.365,-177.581,8.012,148.845
C03325=1140.209,249.883,-68.337,-177.584,8.009,148.845
C03326=1140.213,249.634,-68.309,-177.587,8.006,148.845
C03327=1140.217,249.386,-68.282,-177.589,8.003,148.845
C03328=1140.222,249.138,-68.255,-177.592,8.000,148.845
C03329=1140.226,248.888,-68.227,-177.595,7.997,148.845
C03330=1140.231,248.640,-68.199,-177.598,7.994,148.845
C03331=1140.235,248.392,-68.172,-177.601,7.991,148.845
C03332=1140.240,248.144,-68.145,-177.603,7.988,148.845
C03333=1140.244,247.895,-68.117,-177.606,7.985,148.845
C03334=1140.248,247.646,-68.090,-177.609,7.982,148.845
C03335=1140.253,247.399,-68.062,-177.612,7.979,148.845
C03336=1140.257,247.149,-68.035,-177.615,7.976,148.845
C03337=1140.261,246.901,-68.007,-177.617,7.973,148.845
C03338=1140.266,246.653,-67.980,-177.620,7.970,148.845
C03339=1140.270,246.404,-67.953,-177.623,7.967,148.845
C03340=1140.275,246.156,-67.926,-177.626,7.965,148.845
C03341=1140.279,245.907,-67.898,-177.629,7.962,148.846
C03342=1140.283,245.659,-67.871,-177.631,7.959,148.846
C03343=1140.288,245.410,-67.844,-177.634,7.956,148.846
C03344=1140.293,245.162,-67.817,-177.636,7.953,148.846
C03345=1140.296,244.913,-67.788,-177.639,7.950,148.846
C03346=1140.301,244.665,-67.761,-177.642,7.947,148.846
C03347=1140.305,244.417,-67.735,-177.645,7.944,148.846
C03348=1140.310,244.168,-67.708,-177.648,7.941,148.846
C03349=1140.314,243.920,-67.681,-177.650,7.938,148.846
C03350=1140.318,243.671,-67.653,-177.653,7.935,148.846
C03351=1140.323,243.423,-67.626,-177.656,7.932,148.846
C03352=1140.327,243.174,-67.599,-177.659,7.929,148.846
C03353=1140.332,242.926,-67.571,-177.662,7.926,148.846
C03354=1140.336,242.677,-67.545,-177.664,7.923,148.846
C03355=1140.341,242.429,-67.518,-177.667,7.920,148.846
C03356=1140.345,242.180,-67.490,-177.670,7.918,148.847
C03357=1140.349,241.931,-67.463,-177.673,7.915,148.847
C03358=1140.354,241.683,-67.436,-177.676,7.912,148.847
C03359=1140.358,241.435,-67.410,-177.678,7.909,148.847
C03360=1140.363,241.186,-67.383,-177.681,7.906,148.847
C03361=1140.367,240.938,-67.356,-177.684,7.903,148.847
C03362=1140.372,240.689,-67.329,-177.687,7.900,148.847
C03363=1140.375,240.440,-67.302,-177.690,7.897,148.847
C03364=1140.380,240.192,-67.275,-177.692,7.894,148.847
C03365=1140.385,239.943,-67.248,-177.695,7.891,148.847
C03366=1140.389,239.695,-67.221,-177.698,7.888,148.847
C03367=1140.393,239.447,-67.194,-177.701,7.886,148.847
C03368=1140.398,239.198,-67.167,-177.703,7.883,148.847
C03369=1140.402,238.950,-67.140,-177.706,7.881,148.848
C03370=1140.406,238.701,-67.114,-177.709,7.878,148.848
C03371=1140.411,238.453,-67.087,-177.711,7.875,148.848
C03372=1140.416,238.204,-67.060,-177.714,7.872,148.848
C03373=1140.420,237.956,-67.034,-177.717,7.869,148.848
C03374=1140.425,237.707,-67.007,-177.720,7.866,148.848
C03375=1140.429,237.459,-66.980,-177.723,7.863,148.848
C03376=1140.433,237.210,-66.953,-177.726,7.860,148.848
C03377=1140.437,236.961,-66.926,-177.729,7.858,148.848
C03378=1140.441,236.712,-66.900,-177.731,7.855,148.849
C03379=1140.446,236.464,-66.873,-177.734,7.852,148.849
C03380=1140.451,236.215,-66.846,-177.737,7.849,148.849
C03381=1140.455,235.967,-66.819,-177.740,7.846,148.849
C03382=1140.460,235.695,-66.791,-177.743,7.843,148.849
C03383=1140.465,235.423,-66.761,-177.745,7.840,148.849
C03384=1140.469,235.151,-66.732,-177.749,7.836,148.849
C03385=1140.474,234.880,-66.703,-177.752,7.833,148.849
C03386=1140.479,234.631,-66.677,-177.754,7.830,148.849
C03387=1140.483,234.382,-66.650,-177.758,7.828,148.849
C03388=1140.488,234.134,-66.623,-177.761,7.825,148.850
C03389=1140.492,233.885,-66.597,-177.763,7.822,148.850
C03390=1140.496,233.637,-66.570,-177.766,7.819,148.850
C03391=1140.501,233.388,-66.545,-177.769,7.816,148.850
C03392=1140.505,233.139,-66.517,-177.771,7.814,148.850
C03393=1140.509,232.891,-66.491,-177.774,7.811,148.850
C03394=1140.514,232.642,-66.465,-177.777,7.808,148.850
C03395=1140.519,232.395,-66.439,-177.780,7.805,148.850
C03396=1140.524,232.145,-66.412,-177.782,7.803,148.850
C03397=1140.528,231.897,-66.386,-177.785,7.800,148.850
C03398=1140.532,231.649,-66.360,-177.788,7.797,148.850
C03399=1140.537,231.400,-66.333,-177.791,7.794,148.851
C03400=1140.541,231.151,-66.307,-177.794,7.791,148.851
C03401=1140.545,230.903,-66.280,-177.797,7.788,148.851
C03402=1140.550,230.654,-66.254,-177.800,7.785,148.851
C03403=1140.554,230.405,-66.229,-177.802,7.783,148.851
C03404=1140.559,230.157,-66.202,-177.805,7.780,148.851
C03405=1140.563,229.908,-66.176,-177.807,7.777,148.851
C03406=1140.568,229.660,-66.149,-177.810,7.775,148.851
C03407=1140.572,229.411,-66.123,-177.813,7.772,148.851
C03408=1140.576,229.162,-66.098,-177.816,7.769,148.852
C03409=1140.581,228.914,-66.071,-177.819,7.766,148.852
C03410=1140.585,228.665,-66.045,-177.822,7.763,148.852
C03411=1140.590,228.416,-66.019,-177.825,7.760,148.852
C03412=1140.593,228.168,-65.993,-177.827,7.758,148.852
C03413=1140.599,227.920,-65.967,-177.830,7.755,148.852
C03414=1140.603,227.671,-65.941,-177.832,7.752,148.852
C03415=1140.607,227.423,-65.914,-177.835,7.750,148.852
C03416=1140.612,227.174,-65.888,-177.838,7.747,148.852
C03417=1140.616,226.925,-65.862,-177.841,7.744,148.853
C03418=1140.621,226.676,-65.837,-177.844,7.741,148.853
C03419=1140.625,226.429,-65.810,-177.847,7.738,148.853
C03420=1140.630,226.179,-65.784,-177.849,7.736,148.853
C03421=1140.634,225.931,-65.758,-177.852,7.733,148.853
C03422=1140.639,225.682,-65.733,-177.855,7.730,148.853
C03423=1140.643,225.434,-65.707,-177.858,7.727,148.853
C03424=1140.647,225.185,-65.681,-177.861,7.725,148.854
C03425=1140.652,224.936,-65.654,-177.864,7.722,148.854
C03426=1140.656,224.688,-65.629,-177.866,7.719,148.854
C03427=1140.661,224.439,-65.603,-177.869,7.717,148.854
C03428=1140.666,224.191,-65.577,-177.871,7.714,148.854
C03429=1140.670,223.942,-65.552,-177.874,7.711,148.854
C03430=1140.675,223.693,-65.525,-177.878,7.709,148.854
C03431=1140.679,223.444,-65.500,-177.880,7.706,148.855
C03432=1140.684,223.196,-65.474,-177.883,7.703,148.855
C03433=1140.688,222.947,-65.449,-177.886,7.700,148.855
C03434=1140.692,222.698,-65.423,-177.888,7.698,148.855
C03435=1140.697,222.450,-65.397,-177.891,7.695,148.855
C03436=1140.701,222.201,-65.372,-177.894,7.692,148.855
C03437=1140.705,221.953,-65.346,-177.897,7.689,148.855
C03438=1140.710,221.704,-65.320,-177.900,7.686,148.855
C03439=1140.715,221.456,-65.295,-177.903,7.683,148.856
C03440=1140.719,221.206,-65.268,-177.905,7.681,148.856
C03441=1140.724,220.958,-65.243,-177.908,7.679,148.856
C03442=1140.729,220.710,-65.217,-177.911,7.676,148.856
C03443=1140.733,220.461,-65.192,-177.914,7.673,148.856
C03444=1140.737,220.212,-65.166,-177.917,7.670,148.856
C03445=1140.742,219.964,-65.140,-177.919,7.667,148.856
C03446=1140.746,219.715,-65.115,-177.922,7.665,148.857
C03447=1140.750,219.466,-65.089,-177.925,7.663,148.857
C03448=1140.755,219.218,-65.064,-177.928,7.660,148.857
C03449=1140.760,218.969,-65.038,-177.930,7.657,148.857
C03450=1140.764,218.720,-65.013,-177.934,7.654,148.857
C03451=1140.769,218.472,-64.987,-177.936,7.652,148.857
C03452=1140.773,218.223,-64.962,-177.939,7.649,148.858
C03453=1140.777,217.974,-64.937,-177.942,7.646,148.858
C03454=1140.782,217.726,-64.912,-177.944,7.643,148.858
C03455=1140.786,217.477,-64.886,-177.948,7.641,148.858
C03456=1140.791,217.229,-64.861,-177.950,7.639,148.858
C03457=1140.795,216.979,-64.836,-177.953,7.636,148.858
C03458=1140.799,216.731,-64.810,-177.955,7.633,148.858
C03459=1140.804,216.483,-64.784,-177.959,7.630,148.859
C03460=1140.809,216.233,-64.759,-177.961,7.627,148.859
C03461=1140.813,215.985,-64.734,-177.964,7.625,148.859
C03462=1140.818,215.736,-64.708,-177.967,7.622,148.859
C03463=1140.822,215.487,-64.683,-177.970,7.620,148.859
C03464=1140.826,215.239,-64.658,-177.973,7.617,148.859
C03465=1140.831,214.990,-64.633,-177.975,7.614,148.859
C03466=1140.836,214.741,-64.608,-177.978,7.612,148.860
C03467=1140.840,214.493,-64.582,-177.981,7.609,148.860
C03468=1140.845,214.244,-64.558,-177.984,7.606,148.860
C03469=1140.849,213.995,-64.532,-177.986,7.604,148.860
C03470=1140.853,213.747,-64.507,-177.989,7.601,148.860
C03471=1140.858,213.498,-64.482,-177.992,7.599,148.861
C03472=1140.863,213.250,-64.457,-177.995,7.596,148.861
C03473=1140.867,213.000,-64.432,-177.998,7.593,148.861
C03474=1140.871,212.753,-64.407,-178.001,7.591,148.861
C03475=1140.876,212.503,-64.382,-178.003,7.588,148.861
C03476=1140.881,212.255,-64.356,-178.006,7.586,148.861
C03477=1140.885,212.006,-64.331,-178.009,7.583,148.861
C03478=1140.889,211.758,-64.307,-178.012,7.580,148.862
C03479=1140.894,211.508,-64.282,-178.014,7.578,148.862
C03480=1140.899,211.260,-64.257,-178.017,7.575,148.862
C03481=1140.903,211.011,-64.231,-178.020,7.573,148.862
C03482=1140.908,210.762,-64.207,-178.023,7.570,148.862
C03483=1140.912,210.514,-64.181,-178.025,7.568,148.862
C03484=1140.917,210.265,-64.157,-178.028,7.565,148.863
C03485=1140.921,210.016,-64.132,-178.031,7.562,148.863
C03486=1140.927,209.745,-64.105,-178.034,7.559,148.863
C03487=1140.931,209.474,-64.078,-178.037,7.557,148.863
C03488=1140.936,209.204,-64.051,-178.040,7.554,148.863
C03489=1140.941,208.933,-64.024,-178.044,7.551,148.864
C03490=1140.946,208.685,-63.999,-178.046,7.548,148.864
C03491=1140.950,208.436,-63.974,-178.049,7.545,148.864
C03492=1140.955,208.188,-63.949,-178.052,7.544,148.864
C03493=1140.959,207.938,-63.924,-178.055,7.541,148.864
C03494=1140.963,207.690,-63.900,-178.057,7.538,148.865
C03495=1140.968,207.442,-63.875,-178.060,7.536,148.865
C03496=1140.972,207.192,-63.851,-178.063,7.533,148.865
C03497=1140.977,206.944,-63.826,-178.066,7.530,148.865
C03498=1140.981,206.695,-63.801,-178.069,7.528,148.865
C03499=1140.986,206.447,-63.776,-178.071,7.526,148.866
C03500=1140.991,206.198,-63.751,-178.074,7.523,148.866
C03501=1140.995,205.949,-63.727,-178.077,7.520,148.866
C03502=1141.000,205.700,-63.702,-178.080,7.518,148.866
C03503=1141.004,205.452,-63.678,-178.082,7.515,148.866
C03504=1141.009,205.202,-63.653,-178.086,7.513,148.867
C03505=1141.013,204.954,-63.629,-178.088,7.510,148.867
C03506=1141.018,204.705,-63.604,-178.091,7.508,148.867
C03507=1141.022,204.456,-63.579,-178.094,7.505,148.867
C03508=1141.027,204.208,-63.555,-178.097,7.502,148.867
C03509=1141.031,203.959,-63.531,-178.099,7.500,148.867
C03510=1141.036,203.710,-63.506,-178.102,7.497,148.868
C03511=1141.040,203.462,-63.481,-178.105,7.495,148.868
C03512=1141.045,203.213,-63.457,-178.108,7.493,148.868
C03513=1141.049,202.964,-63.432,-178.111,7.490,148.868
C03514=1141.054,202.715,-63.408,-178.113,7.487,148.868
C03515=1141.059,202.467,-63.384,-178.116,7.485,148.869
C03516=1141.063,202.218,-63.359,-178.119,7.482,148.869
C03517=1141.068,201.968,-63.335,-178.122,7.480,148.869
C03518=1141.072,201.720,-63.311,-178.125,7.477,148.869
C03519=1141.077,201.471,-63.287,-178.127,7.475,148.869
C03520=1141.081,201.222,-63.262,-178.130,7.472,148.870
C03521=1141.086,200.973,-63.238,-178.133,7.469,148.870
C03522=1141.090,200.725,-63.214,-178.136,7.468,148.870
C03523=1141.095,200.476,-63.189,-178.139,7.465,148.870
C03524=1141.099,200.227,-63.165,-178.142,7.462,148.870
C03525=1141.103,199.979,-63.141,-178.144,7.460,148.871
C03526=1141.109,199.729,-63.117,-178.147,7.457,148.871
C03527=1141.113,199.481,-63.093,-178.150,7.455,148.871
C03528=1141.118,199.233,-63.069,-178.153,7.453,148.871
C03529=1141.122,198.983,-63.044,-178.155,7.450,148.871
C03530=1141.127,198.735,-63.019,-178.158,7.448,148.872
C03531=1141.131,198.486,-62.996,-178.161,7.445,148.872
C03532=1141.136,198.237,-62.972,-178.164,7.442,148.872
C03533=1141.141,197.989,-62.947,-178.166,7.440,148.872
C03534=1141.145,197.739,-62.923,-178.170,7.438,148.873
C03535=1141.149,197.490,-62.900,-178.172,7.435,148.873
C03536=1141.154,197.242,-62.875,-178.175,7.433,148.873
C03537=1141.159,196.993,-62.851,-178.178,7.430,148.873
C03538=1141.164,196.744,-62.827,-178.181,7.427,148.873
C03539=1141.167,196.495,-62.803,-178.183,7.426,148.874
C03540=1141.172,196.247,-62.779,-178.186,7.423,148.874
C03541=1141.176,195.998,-62.756,-178.190,7.420,148.874
C03542=1141.182,195.749,-62.731,-178.192,7.418,148.874
C03543=1141.186,195.500,-62.708,-178.195,7.416,148.875
C03544=1141.191,195.252,-62.683,-178.197,7.413,148.875
C03545=1141.195,195.003,-62.659,-178.201,7.411,148.875
C03546=1141.199,194.753,-62.636,-178.203,7.408,148.875
C03547=1141.204,194.505,-62.612,-178.206,7.406,148.876
C03548=1141.209,194.256,-62.588,-178.209,7.403,148.876
C03549=1141.213,194.007,-62.564,-178.211,7.401,148.876
C03550=1141.218,193.758,-62.540,-178.214,7.399,148.876
C03551=1141.223,193.510,-62.516,-178.217,7.396,148.876
C03552=1141.227,193.261,-62.493,-178.220,7.394,148.877
C03553=1141.232,193.012,-62.469,-178.223,7.391,148.877
C03554=1141.236,192.763,-62.445,-178.226,7.389,148.877
C03555=1141.241,192.515,-62.421,-178.228,7.387,148.877
C03556=1141.245,192.266,-62.398,-178.231,7.384,148.877
C03557=1141.251,192.017,-62.373,-178.234,7.382,148.878
C03558=1141.255,191.767,-62.350,-178.237,7.379,148.878
C03559=1141.259,191.518,-62.326,-178.240,7.376,148.878
C03560=1141.264,191.270,-62.302,-178.242,7.375,148.878
C03561=1141.268,191.021,-62.279,-178.245,7.372,148.879
C03562=1141.273,190.773,-62.255,-178.248,7.370,148.879
C03563=1141.278,190.523,-62.231,-178.251,7.367,148.879
C03564=1141.282,190.274,-62.208,-178.253,7.365,148.879
C03565=1141.287,190.026,-62.184,-178.256,7.363,148.879
C03566=1141.291,189.777,-62.160,-178.260,7.360,148.880
C03567=1141.296,189.528,-62.137,-178.262,7.358,148.880
C03568=1141.301,189.279,-62.114,-178.265,7.355,148.880
C03569=1141.305,189.031,-62.090,-178.267,7.353,148.880
C03570=1141.310,188.781,-62.066,-178.271,7.351,148.881
C03571=1141.315,188.532,-62.043,-178.273,7.348,148.881
C03572=1141.319,188.283,-62.020,-178.276,7.346,148.881
C03573=1141.324,188.035,-61.996,-178.279,7.343,148.881
C03574=1141.328,187.786,-61.973,-178.282,7.342,148.882
C03575=1141.332,187.537,-61.949,-178.285,7.339,148.882
C03576=1141.337,187.288,-61.926,-178.287,7.337,148.882
C03577=1141.342,187.039,-61.903,-178.290,7.334,148.883
C03578=1141.347,186.791,-61.879,-178.293,7.332,148.883
C03579=1141.351,186.542,-61.856,-178.296,7.330,148.883
C03580=1141.356,186.293,-61.832,-178.299,7.327,148.883
C03581=1141.361,186.044,-61.809,-178.301,7.325,148.884
C03582=1141.365,185.796,-61.786,-178.304,7.322,148.884
C03583=1141.369,185.547,-61.763,-178.307,7.320,148.884
C03584=1141.374,185.298,-61.739,-178.310,7.318,148.884
C03585=1141.379,185.049,-61.716,-178.312,7.316,148.884
C03586=1141.383,184.800,-61.692,-178.316,7.313,148.885
C03587=1141.388,184.551,-61.669,-178.318,7.311,148.885
C03588=1141.392,184.302,-61.646,-178.321,7.309,148.885
C03589=1141.397,184.053,-61.623,-178.323,7.307,148.885
C03590=1141.402,183.784,-61.597,-178.327,7.304,148.886
C03591=1141.407,183.514,-61.572,-178.330,7.301,148.886
C03592=1141.413,183.244,-61.547,-178.333,7.299,148.886
C03593=1141.417,182.975,-61.522,-178.336,7.296,148.887
C03594=1141.422,182.726,-61.499,-178.339,7.294,148.887
C03595=1141.427,182.477,-61.476,-178.342,7.291,148.887
C03596=1141.431,182.228,-61.453,-178.344,7.290,148.887
C03597=1141.435,181.979,-61.430,-178.347,7.287,148.888
C03598=1141.440,181.730,-61.407,-178.350,7.285,148.888
C03599=1141.445,181.481,-61.384,-178.353,7.283,148.888
C03600=1141.449,181.233,-61.361,-178.355,7.280,148.888
C03601=1141.454,180.984,-61.338,-178.359,7.278,148.889
C03602=1141.459,180.735,-61.314,-178.361,7.276,148.889
C03603=1141.462,180.486,-61.292,-178.364,7.273,148.889
C03604=1141.468,180.236,-61.269,-178.367,7.272,148.890
C03605=1141.473,179.988,-61.246,-178.370,7.269,148.890
C03606=1141.477,179.739,-61.223,-178.372,7.267,148.890
C03607=1141.481,179.490,-61.200,-178.375,7.264,148.890
C03608=1141.486,179.241,-61.176,-178.378,7.262,148.891
C03609=1141.490,178.992,-61.154,-178.381,7.260,148.891
C03610=1141.496,178.743,-61.131,-178.383,7.258,148.891
C03611=1141.500,178.495,-61.109,-178.387,7.255,148.891
C03612=1141.504,178.246,-61.085,-178.389,7.253,148.892
C03613=1141.509,177.996,-61.063,-178.392,7.251,148.892
C03614=1141.514,177.748,-61.040,-178.395,7.249,148.892
C03615=1141.519,177.499,-61.017,-178.398,7.246,148.892
C03616=1141.523,177.250,-60.994,-178.400,7.244,148.893
C03617=1141.528,177.001,-60.971,-178.404,7.242,148.893
C03618=1141.532,176.753,-60.949,-178.406,7.240,148.893
C03619=1141.537,176.504,-60.926,-178.409,7.237,148.894
C03620=1141.542,176.254,-60.903,-178.411,7.235,148.894
C03621=1141.546,176.005,-60.880,-178.415,7.232,148.894
C03622=1141.551,175.756,-60.858,-178.417,7.231,148.894
C03623=1141.555,175.508,-60.835,-178.420,7.228,148.895
C03624=1141.560,175.259,-60.812,-178.423,7.226,148.895
C03625=1141.565,175.010,-60.790,-178.426,7.224,148.895
C03626=1141.570,174.761,-60.767,-178.428,7.221,148.895
C03627=1141.574,174.512,-60.745,-178.431,7.220,148.896
C03628=1141.579,174.262,-60.721,-178.434,7.217,148.896
C03629=1141.584,174.014,-60.700,-178.437,7.215,148.896
C03630=1141.587,173.765,-60.677,-178.440,7.213,148.897
C03631=1141.593,173.515,-60.654,-178.443,7.211,148.897
C03632=1141.597,173.267,-60.632,-178.445,7.208,148.897
C03633=1141.602,173.018,-60.609,-178.448,7.206,148.898
C03634=1141.606,172.769,-60.587,-178.451,7.204,148.898
C03635=1141.612,172.520,-60.564,-178.454,7.202,148.898
C03636=1141.616,172.271,-60.542,-178.457,7.199,148.898
C03637=1141.620,172.023,-60.520,-178.460,7.197,148.899
C03638=1141.625,171.774,-60.496,-178.462,7.195,148.899
C03639=1141.629,171.524,-60.474,-178.465,7.193,148.899
C03640=1141.635,171.275,-60.452,-178.468,7.191,148.900
C03641=1141.639,171.027,-60.429,-178.471,7.188,148.900
C03642=1141.643,170.777,-60.407,-178.473,7.186,148.900
C03643=1141.649,170.529,-60.384,-178.477,7.184,148.900
C03644=1141.653,170.280,-60.362,-178.479,7.182,148.901
C03645=1141.658,170.031,-60.341,-178.482,7.180,148.901
C03646=1141.662,169.782,-60.317,-178.485,7.178,148.901
C03647=1141.667,169.533,-60.295,-178.487,7.175,148.902
